FUNCTION_BLOCK "SysPos"   // FB2010, FBD
TITLE = manage a standard positioning system
{ S7_Optimized_Access := 'TRUE' }
AUTHOR : MiCROTEC
VERSION : 1.2
// -2017.03 : Martin
// stored: AutoNumber false, MemoryReserve 100, SetENOAutomatically false
   VAR_INPUT
      actual { ExternalAccessible := 'False'; ExternalVisible := 'False'; ExternalWritable := 'False'} : Real;   // actual position
      target { ExternalAccessible := 'False'; ExternalVisible := 'False'; ExternalWritable := 'False'} : Real;   // target position , start new position only if target position change
      tarMinPos { ExternalAccessible := 'False'; ExternalVisible := 'False'; ExternalWritable := 'False'} : Real;   // target position minimum
      tarMaxPos { ExternalAccessible := 'False'; ExternalVisible := 'False'; ExternalWritable := 'False'} : Real;   // target position maximum
      tolerance { ExternalAccessible := 'False'; ExternalVisible := 'False'; ExternalWritable := 'False'} : Real;   // tolerance for output signal position ok
      regPoint { ExternalAccessible := 'False'; ExternalVisible := 'False'; ExternalWritable := 'False'} : Real;   // regulation point (stop point before target position)
      regOn { ExternalAccessible := 'False'; ExternalVisible := 'False'; ExternalWritable := 'False'} : Bool;   // continuouse regulation on
      restart { ExternalAccessible := 'False'; ExternalVisible := 'False'; ExternalWritable := 'False'} : Bool;   // restart new positioning
      auto { ExternalAccessible := 'False'; ExternalVisible := 'False'; ExternalWritable := 'False'} : Bool;   // automatic (manP/manM and gain works only if auto is on)
      manP { ExternalAccessible := 'False'; ExternalVisible := 'False'; ExternalWritable := 'False'} : Bool;   // manual button plus
      manM { ExternalAccessible := 'False'; ExternalVisible := 'False'; ExternalWritable := 'False'} : Bool;   // manual button minus
      manPValue { ExternalAccessible := 'False'; ExternalVisible := 'False'; ExternalWritable := 'False'} : Real := 10.0;   // increase value in hand mode
      manMValue { ExternalAccessible := 'False'; ExternalVisible := 'False'; ExternalWritable := 'False'} : Real := 10.0;   // decrease value in hand mode
      stopRamp { ExternalAccessible := 'False'; ExternalVisible := 'False'; ExternalWritable := 'False'} : Real;   // position for stopramp
      stopSpeed { ExternalAccessible := 'False'; ExternalVisible := 'False'; ExternalWritable := 'False'} : Real;   // minimum speed for stopramp [0.0-1.0]
      approachPoint { ExternalAccessible := 'False'; ExternalVisible := 'False'; ExternalWritable := 'False'} : Real;   // aproach point, if its 0 than its OFF
   END_VAR
   VAR_OUTPUT
      plus { ExternalAccessible := 'False'; ExternalVisible := 'False'; ExternalWritable := 'False'} : Bool;   // command plus
      minus { ExternalAccessible := 'False'; ExternalVisible := 'False'; ExternalWritable := 'False'} : Bool;   // command minus
      slow { ExternalAccessible := 'False'; ExternalVisible := 'False'; ExternalWritable := 'False'} : Bool;   // slow
      posOk { ExternalAccessible := 'False'; ExternalVisible := 'False'; ExternalWritable := 'False'} : Bool;   // position ok
      tar { ExternalAccessible := 'False'; ExternalVisible := 'False'; ExternalWritable := 'False'} : Real;   // target position
      speedGain { ExternalAccessible := 'False'; ExternalVisible := 'False'; ExternalWritable := 'False'} : Real;   // gain for speed regulation ["StopSpeed" to 1.0]
   END_VAR
   VAR_IN_OUT
      Enc : "TypeEncoder";
   END_VAR
   VAR
      var { ExternalAccessible := 'False'; ExternalVisible := 'False'; ExternalWritable := 'False'} : Struct
         "bool" : Bool;
         "byte" : Byte;
         "word" : Word;
         "dword" : DWord;
         "int" : Int;
         "dint" : DInt;
         "real" : Real;
         s5time : S5Time;
         "time" : Time;
         hm : Array[1..16] of Bool;
         fm : Array[1..16] of Bool;
      END_STRUCT;
      statTargetOld { ExternalAccessible := 'False'; ExternalVisible := 'False'; ExternalWritable := 'False'} : Real;
      statApproachPoint { ExternalAccessible := 'False'; ExternalVisible := 'False'; ExternalWritable := 'False'} : Real;
      statRegPlusPos { ExternalAccessible := 'False'; ExternalVisible := 'False'; ExternalWritable := 'False'} : Real;
      statRegMinusPos { ExternalAccessible := 'False'; ExternalVisible := 'False'; ExternalWritable := 'False'} : Real;
      statInTolerance { ExternalAccessible := 'False'; ExternalVisible := 'False'; ExternalWritable := 'False'} : Bool;
      statAproachRun { ExternalAccessible := 'False'; ExternalVisible := 'False'; ExternalWritable := 'False'} : Bool;
      StatPosOk { ExternalAccessible := 'False'; ExternalVisible := 'False'; ExternalWritable := 'False'} : Bool;
      statSpeedDelta { ExternalAccessible := 'False'; ExternalVisible := 'False'; ExternalWritable := 'False'} : Real;
      statSpeedPerMm { ExternalAccessible := 'False'; ExternalVisible := 'False'; ExternalWritable := 'False'} : Real;
      statTarMin { ExternalAccessible := 'False'; ExternalVisible := 'False'; ExternalWritable := 'False'} : Bool;
      statTarMax { ExternalAccessible := 'False'; ExternalVisible := 'False'; ExternalWritable := 'False'} : Bool;
      statTar { ExternalAccessible := 'False'; ExternalVisible := 'False'; ExternalWritable := 'False'} : Real;
      statPlus { ExternalAccessible := 'False'; ExternalVisible := 'False'; ExternalWritable := 'False'} : Bool;
      statMinus { ExternalAccessible := 'False'; ExternalVisible := 'False'; ExternalWritable := 'False'} : Bool;
      statSpeedGain { ExternalAccessible := 'False'; ExternalVisible := 'False'; ExternalWritable := 'False'} : Real;
      statSlow { ExternalAccessible := 'False'; ExternalVisible := 'False'; ExternalWritable := 'False'} : Bool;
      statTarMaxPosOld : Real;
      statTarMinPosOld : Real;
   END_VAR
   VAR_TEMP   // added for the SCL form of the ladder/FBD networks
      _w1 : Bool;
      _w2 : Bool;
      _w3 : Bool;
   END_VAR
BEGIN

REGION Network 1: manual change target position
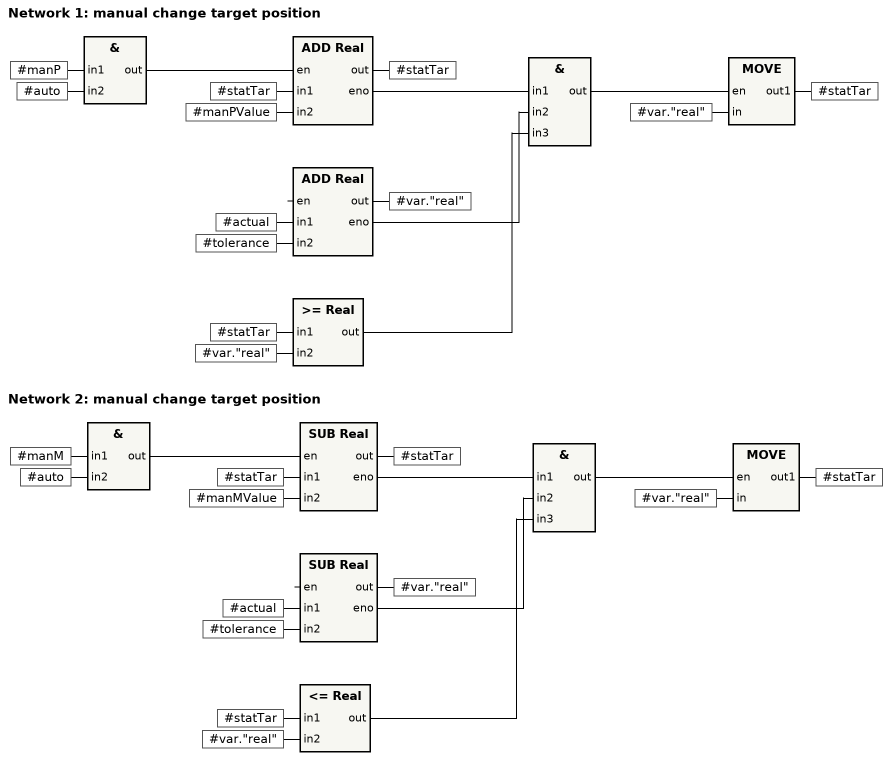
   // ENO of a box is taken as its EN; it also drops when the box reports an error
   #_w1 := #manP AND #auto;
   IF #_w1 THEN #statTar := #statTar + #manPValue; END_IF;
   #var."real" := #actual + #tolerance;
   IF #_w1 AND (#statTar >= #var."real") THEN #statTar := #var."real"; END_IF;
END_REGION

REGION Network 2: manual change target position
   // ENO of a box is taken as its EN; it also drops when the box reports an error
   #_w1 := #manM AND #auto;
   IF #_w1 THEN #statTar := #statTar - #manMValue; END_IF;
   #var."real" := #actual - #tolerance;
   IF #_w1 AND (#statTar <= #var."real") THEN #statTar := #var."real"; END_IF;
END_REGION

REGION Network 3: start positioning
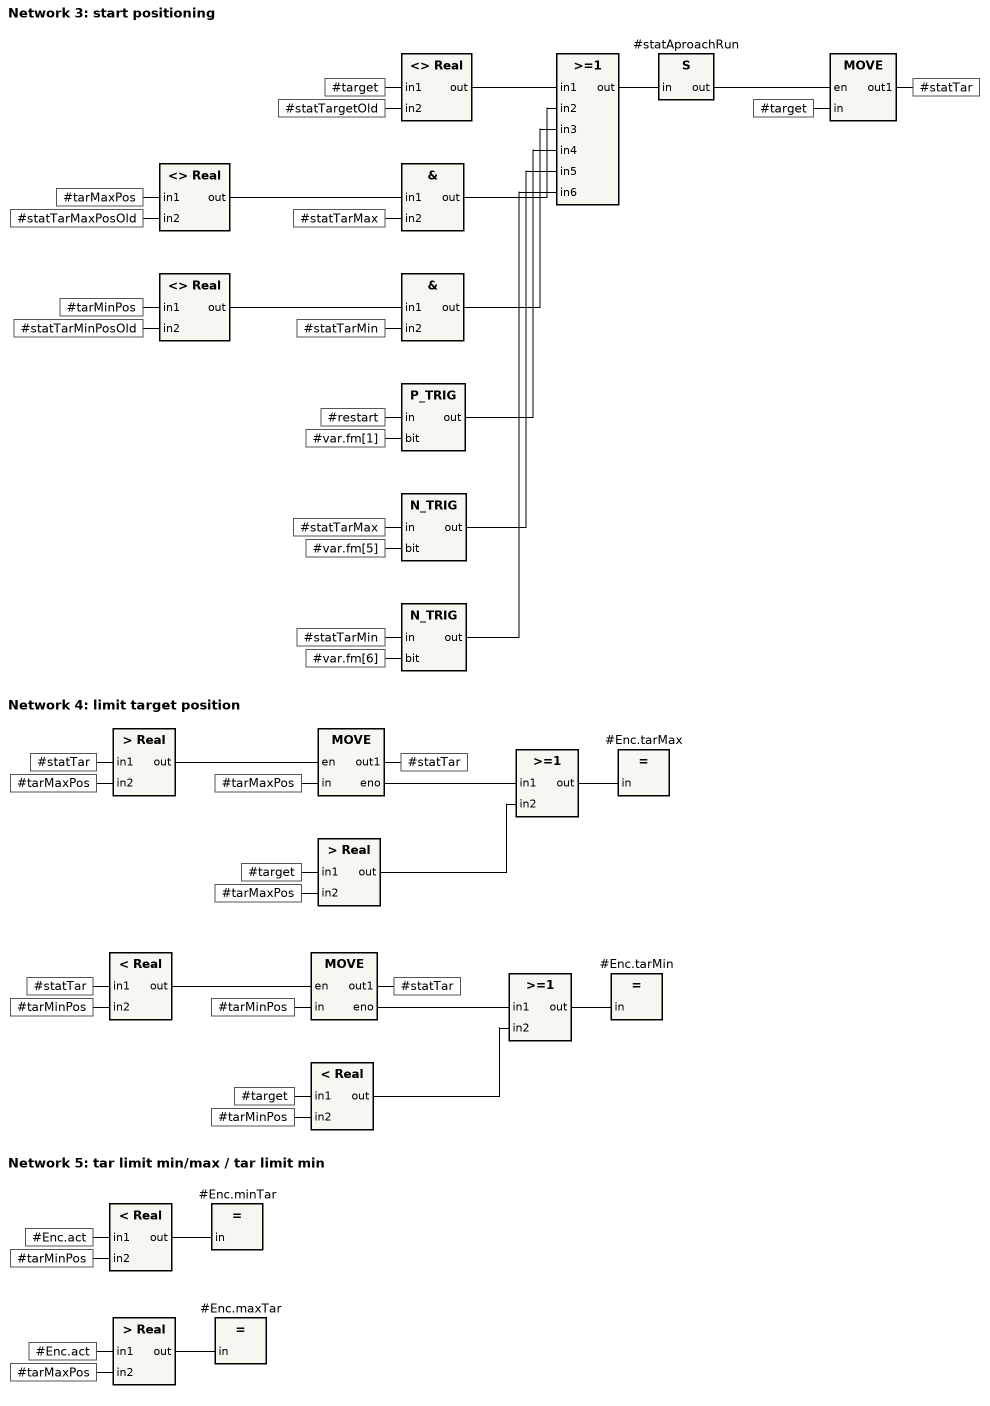
   #_w1 := #restart AND NOT #var.fm[1];   // rising edge
   #var.fm[1] := #restart;
   #_w2 := NOT #statTarMax AND #var.fm[5];   // falling edge
   #var.fm[5] := #statTarMax;
   #_w3 := NOT #statTarMin AND #var.fm[6];   // falling edge
   #var.fm[6] := #statTarMin;
   IF (#target <> #statTargetOld) OR ((#tarMaxPos <> #statTarMaxPosOld) AND #statTarMax) OR ((#tarMinPos <> #statTarMinPosOld) AND #statTarMin) OR #_w1 OR #_w2 OR #_w3 THEN
       #statAproachRun := TRUE;
       #statTar := #target;
   END_IF;
END_REGION

REGION Network 4: limit target position
   // ENO of a box is taken as its EN; it also drops when the box reports an error
   #_w1 := #statTar > #tarMaxPos;
   IF #_w1 THEN #statTar := #tarMaxPos; END_IF;
   #Enc.tarMax := #_w1 OR (#target > #tarMaxPos);
   #_w2 := #statTar < #tarMinPos;
   IF #_w2 THEN #statTar := #tarMinPos; END_IF;
   #Enc.tarMin := #_w2 OR (#target < #tarMinPos);
END_REGION

REGION Network 5: tar limit min/max / tar limit min
   #Enc.minTar := #Enc.act < #tarMinPos;
   #Enc.maxTar := #Enc.act > #tarMaxPos;
END_REGION

REGION Network 6 (SCL): approach/regulation point
   #statApproachPoint := #statTar + #approachPoint;

   #statRegMinusPos := #statTar - #regPoint;
   #statRegPlusPos := #statTar + #regPoint;
END_REGION

REGION Network 7: approachpoint reach
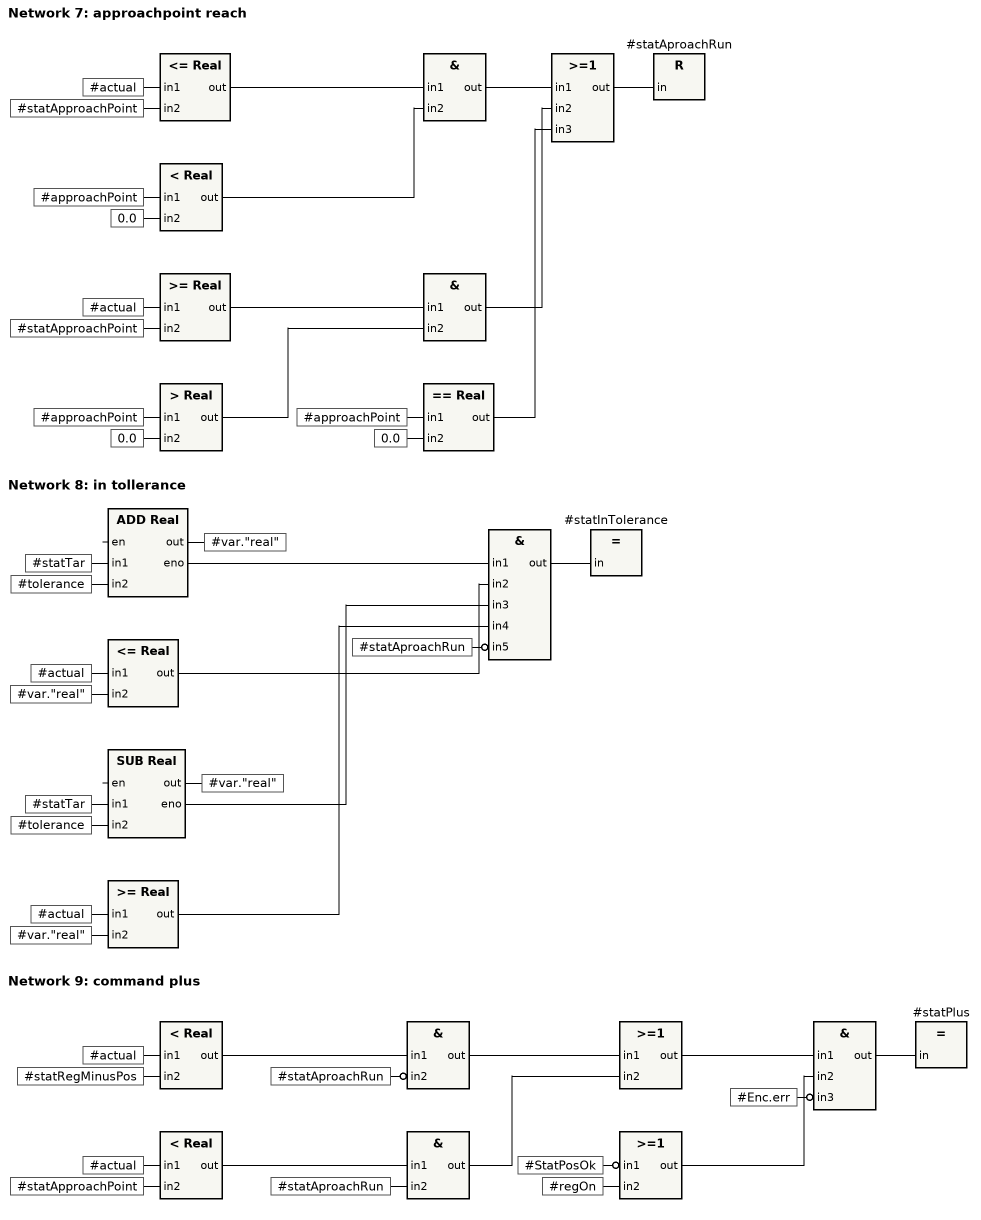
   IF ((#actual <= #statApproachPoint) AND (#approachPoint < 0.0)) OR ((#actual >= #statApproachPoint) AND (#approachPoint > 0.0)) OR (#approachPoint = 0.0) THEN
       #statAproachRun := FALSE;
   END_IF;
END_REGION

REGION Network 8: in tollerance
   // ENO of a box is taken as its EN; it also drops when the box reports an error
   #var."real" := #statTar + #tolerance;
   #_w1 := #actual <= #var."real";
   #var."real" := #statTar - #tolerance;
   #statInTolerance := #_w1 AND (#actual >= #var."real") AND NOT #statAproachRun;
END_REGION

REGION Network 9: command plus
   #statPlus := (((#actual < #statRegMinusPos) AND NOT #statAproachRun) OR ((#actual < #statApproachPoint) AND #statAproachRun)) AND (NOT #StatPosOk OR #regOn) AND NOT #Enc.err;
END_REGION

REGION Network 10: command minus
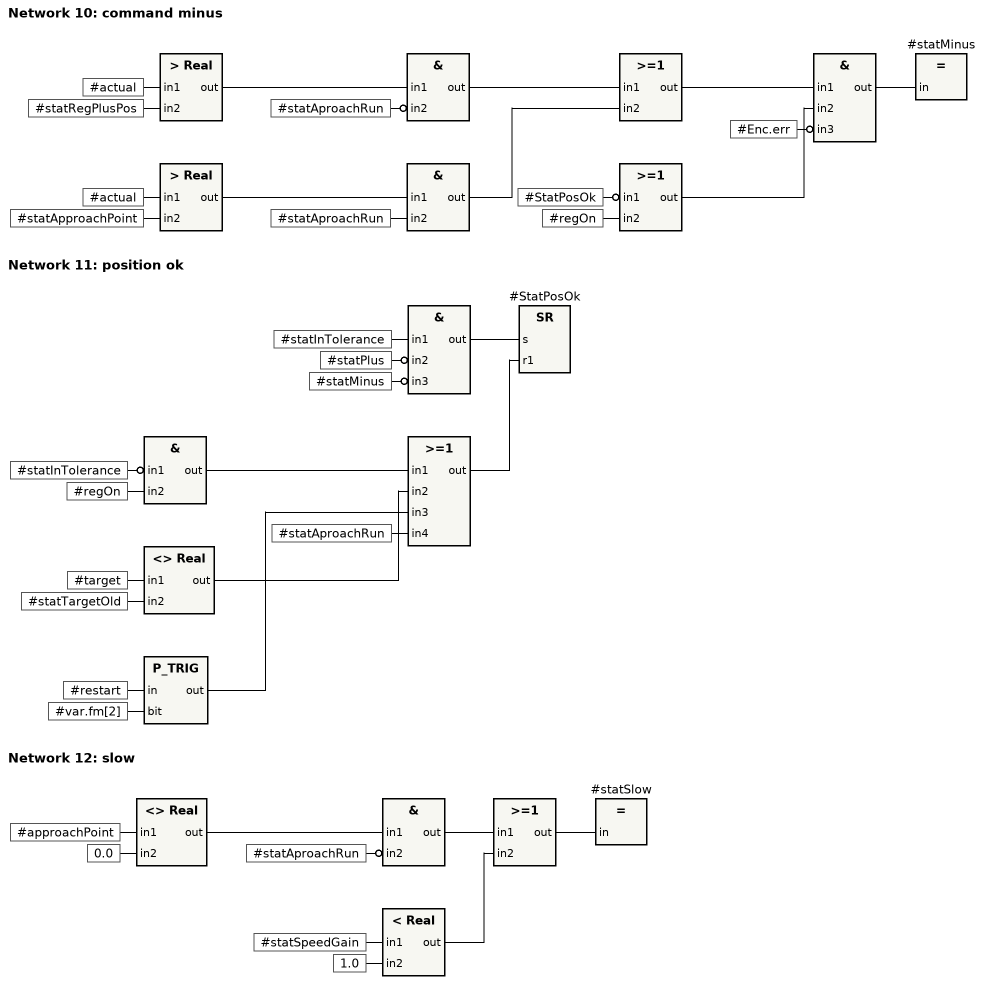
   #statMinus := (((#actual > #statRegPlusPos) AND NOT #statAproachRun) OR ((#actual > #statApproachPoint) AND #statAproachRun)) AND (NOT #StatPosOk OR #regOn) AND NOT #Enc.err;
END_REGION

REGION Network 11: position ok
   #_w1 := #restart AND NOT #var.fm[2];   // rising edge
   #var.fm[2] := #restart;
   IF #statInTolerance AND NOT #statPlus AND NOT #statMinus THEN
       #StatPosOk := TRUE;   // SR flip-flop
   END_IF;
   IF (NOT #statInTolerance AND #regOn) OR (#target <> #statTargetOld) OR #_w1 OR #statAproachRun THEN
       #StatPosOk := FALSE;
   END_IF;
END_REGION

REGION Network 12: slow
   #statSlow := ((#approachPoint <> 0.0) AND NOT #statAproachRun) OR (#statSpeedGain < 1.0);
END_REGION

REGION Network 13 (SCL): old position
   #statTargetOld := #target;
   #statTarMaxPosOld := #tarMaxPos;
   #statTarMinPosOld := #tarMinPos;
END_REGION

REGION Network 14 (SCL): speed gain for stop ramp
   #statSpeedDelta := 1.0 - #stopSpeed;
   #statSpeedPerMm := #statSpeedDelta / #stopRamp;
   #statSpeedGain := #stopSpeed + ABS_REAL((#statTar - #actual) * #statSpeedPerMm);

   IF #statSpeedGain < #stopSpeed THEN
       #statSpeedGain := #stopSpeed;
   END_IF;

   IF #statSpeedGain > 1.0 OR NOT #auto THEN
       #statSpeedGain := 1.0;
   END_IF;
END_REGION

REGION Network 15 (SCL): write outputs
       #plus := #statPlus;
       #minus := #statMinus;
       #slow:= #statSlow;
       #posOk := #StatPosOk;
       #tar := #statTar;
       #speedGain := #statSpeedGain;
END_REGION

REGION Network 16 (SCL): in/out data
       #Enc.tarMinPos := #tarMinPos;
       #Enc.tarMaxPos := #tarMaxPos;
       #Enc.act := #actual;
       #Enc.tar := #statTar;
       #Enc.posOk := #StatPosOk;
END_REGION
END_FUNCTION_BLOCK

FUNCTION_BLOCK "SysMotor"   // FB2060, FBD
TITLE = manage a motor with contactor equipment
{ S7_Optimized_Access := 'TRUE' }
AUTHOR : MiCROTEC
VERSION : 1.6
// -2017.03 : Martin
// stored: AutoNumber false, MemoryReserve 100, SetENOAutomatically false
   VAR_INPUT
      area { ExternalAccessible := 'False'; ExternalVisible := 'False'; ExternalWritable := 'False'} : Bool;   // 1=safety area on
      auto { ExternalAccessible := 'False'; ExternalVisible := 'False'; ExternalWritable := 'False'} : Bool;   // automatic
      manP { ExternalAccessible := 'False'; ExternalVisible := 'False'; ExternalWritable := 'False'} : Bool;   // manual plus
      manM { ExternalAccessible := 'False'; ExternalVisible := 'False'; ExternalWritable := 'False'} : Bool;   // manual minus
      autoP { ExternalAccessible := 'False'; ExternalVisible := 'False'; ExternalWritable := 'False'} : Bool;   // automatic plus
      autoM { ExternalAccessible := 'False'; ExternalVisible := 'False'; ExternalWritable := 'False'} : Bool;   // automatic minus
      ack { ExternalAccessible := 'False'; ExternalVisible := 'False'; ExternalWritable := 'False'} : Bool;   // fault acknowledge
      lampTest { ExternalAccessible := 'False'; ExternalVisible := 'False'; ExternalWritable := 'False'} : Bool;   // lamptest
      enableP { ExternalAccessible := 'False'; ExternalVisible := 'False'; ExternalWritable := 'False'} : Bool;   // release plus
      enableM { ExternalAccessible := 'False'; ExternalVisible := 'False'; ExternalWritable := 'False'} : Bool;   // release minus
      enAutoP { ExternalAccessible := 'False'; ExternalVisible := 'False'; ExternalWritable := 'False'} : Bool;   // release automatic plus
      enAutoM { ExternalAccessible := 'False'; ExternalVisible := 'False'; ExternalWritable := 'False'} : Bool;   // release automatic minus
      mpMotor { ExternalAccessible := 'False'; ExternalVisible := 'False'; ExternalWritable := 'False'} : Bool;   // 1=motor protection switch ok
      mpBrake { ExternalAccessible := 'False'; ExternalVisible := 'False'; ExternalWritable := 'False'} : Bool;   // 1=motor protection switch brake ok
      mpBrake2 { ExternalAccessible := 'False'; ExternalVisible := 'False'; ExternalWritable := 'False'} : Bool;   // 1=motor protection switch brake ok
      mpFan { ExternalAccessible := 'False'; ExternalVisible := 'False'; ExternalWritable := 'False'} : Bool;   // 1=motor protection switch fan ok
      thMotor { ExternalAccessible := 'False'; ExternalVisible := 'False'; ExternalWritable := 'False'} : Bool;   // 1=thermal contact motor ok
      thMotorRtd { ExternalAccessible := 'False'; ExternalVisible := 'False'; ExternalWritable := 'False'} : Int;   // thermal contact motor AE 8xRTD
      mSwitch { ExternalAccessible := 'False'; ExternalVisible := 'False'; ExternalWritable := 'False'} : Bool;   // 1=maintenance switch is ok
      fdb { ExternalAccessible := 'False'; ExternalVisible := 'False'; ExternalWritable := 'False'} : Bool;   // 1=feedback circuit ok
      changeDirTime { ExternalAccessible := 'False'; ExternalVisible := 'False'; ExternalWritable := 'False'} : Time := T#500MS;   // time wait to restart in oder direction
      restartTime { ExternalAccessible := 'False'; ExternalVisible := 'False'; ExternalWritable := 'False'} : Time := T#500MS;   // time wait to restart in any direction
      brakeOnTime { ExternalAccessible := 'False'; ExternalVisible := 'False'; ExternalWritable := 'False'} : Time := T#10MS;   // time wait to open the brake
      brakeOffTime { ExternalAccessible := 'False'; ExternalVisible := 'False'; ExternalWritable := 'False'} : Time := T#10MS;   // time wait to close the brake
      metPerMin { ExternalAccessible := 'False'; ExternalVisible := 'False'; ExternalWritable := 'False'} : Real := 1.0;   // meter per minute with nominal speed
      cycle { ExternalAccessible := 'False'; ExternalVisible := 'False'; ExternalWritable := 'False'} : Real;   // cycle
   END_VAR
   VAR_OUTPUT
      plus { ExternalAccessible := 'False'; ExternalVisible := 'False'; ExternalWritable := 'False'} : Bool;   // drive plus
      minus { ExternalAccessible := 'False'; ExternalVisible := 'False'; ExternalWritable := 'False'} : Bool;   // drive minus
      brake { ExternalAccessible := 'False'; ExternalVisible := 'False'; ExternalWritable := 'False'} : Bool;   // brake open
      brake2 { ExternalAccessible := 'False'; ExternalVisible := 'False'; ExternalWritable := 'False'} : Bool;   // brake open
      enStartP { ExternalAccessible := 'False'; ExternalVisible := 'False'; ExternalWritable := 'False'} : Bool;   // release drive plus
      enStartM { ExternalAccessible := 'False'; ExternalVisible := 'False'; ExternalWritable := 'False'} : Bool;   // release drive minus
      fan { ExternalAccessible := 'False'; ExternalVisible := 'False'; ExternalWritable := 'False'} : Bool;   // fan on
      lamp { ExternalAccessible := 'False'; ExternalVisible := 'False'; ExternalWritable := 'False'} : Bool;   // indication lamp
      lamp2 { ExternalAccessible := 'False'; ExternalVisible := 'False'; ExternalWritable := 'False'} : Bool;   // indication lamp 2
      actSpeed { ExternalAccessible := 'False'; ExternalVisible := 'False'; ExternalWritable := 'False'} : Real;   // actual speed
      mmCycle { ExternalAccessible := 'False'; ExternalVisible := 'False'; ExternalWritable := 'False'} : Real;   // milimeter per cycle
      err { ExternalAccessible := 'False'; ExternalVisible := 'False'; ExternalWritable := 'False'} : Bool;   // fault
   END_VAR
   VAR_IN_OUT
      Mot : "TypeMotor";   // Daten an VISU Motor
   END_VAR
   VAR
      var { ExternalAccessible := 'False'; ExternalVisible := 'False'; ExternalWritable := 'False'} : Struct
         true : Bool;
         false : Bool;
         "bool" : Bool;
         "byte" : Byte;
         "word" : Word;
         "dword" : DWord;
         "int" : Int;
         "dint" : DInt;
         "real" : Real;
         s5time : S5Time;
         "time" : Time;
         hm : Array[1..50] of Bool;
         fm : Array[1..50] of Bool;
      END_STRUCT;
      T { ExternalAccessible := 'False'; ExternalVisible := 'False'; ExternalWritable := 'False'} : Array[1..15] of IEC_TIMER;
      restartBreak { ExternalAccessible := 'False'; ExternalVisible := 'False'; ExternalWritable := 'False'} : Bool;
      man { ExternalAccessible := 'False'; ExternalVisible := 'False'; ExternalWritable := 'False'} : Bool;
      changeDirDelM { ExternalAccessible := 'False'; ExternalVisible := 'False'; ExternalWritable := 'False'} : Bool;
      changeDirDelP { ExternalAccessible := 'False'; ExternalVisible := 'False'; ExternalWritable := 'False'} : Bool;
      mpFanOffDel { ExternalAccessible := 'False'; ExternalVisible := 'False'; ExternalWritable := 'False'} : Bool;
      brakeOnDel { ExternalAccessible := 'False'; ExternalVisible := 'False'; ExternalWritable := 'False'} : Bool;
      brakeOffDel { ExternalAccessible := 'False'; ExternalVisible := 'False'; ExternalWritable := 'False'} : Bool;
      autoOld { ExternalAccessible := 'False'; ExternalVisible := 'False'; ExternalWritable := 'False'} : Bool;
   END_VAR
   VAR_TEMP
      tempAck : Bool;
   END_VAR
   VAR_TEMP   // added for the SCL form of the ladder/FBD networks
      _w1 : Bool;
      _w2 : Bool;
   END_VAR
BEGIN

REGION Network 1: ack
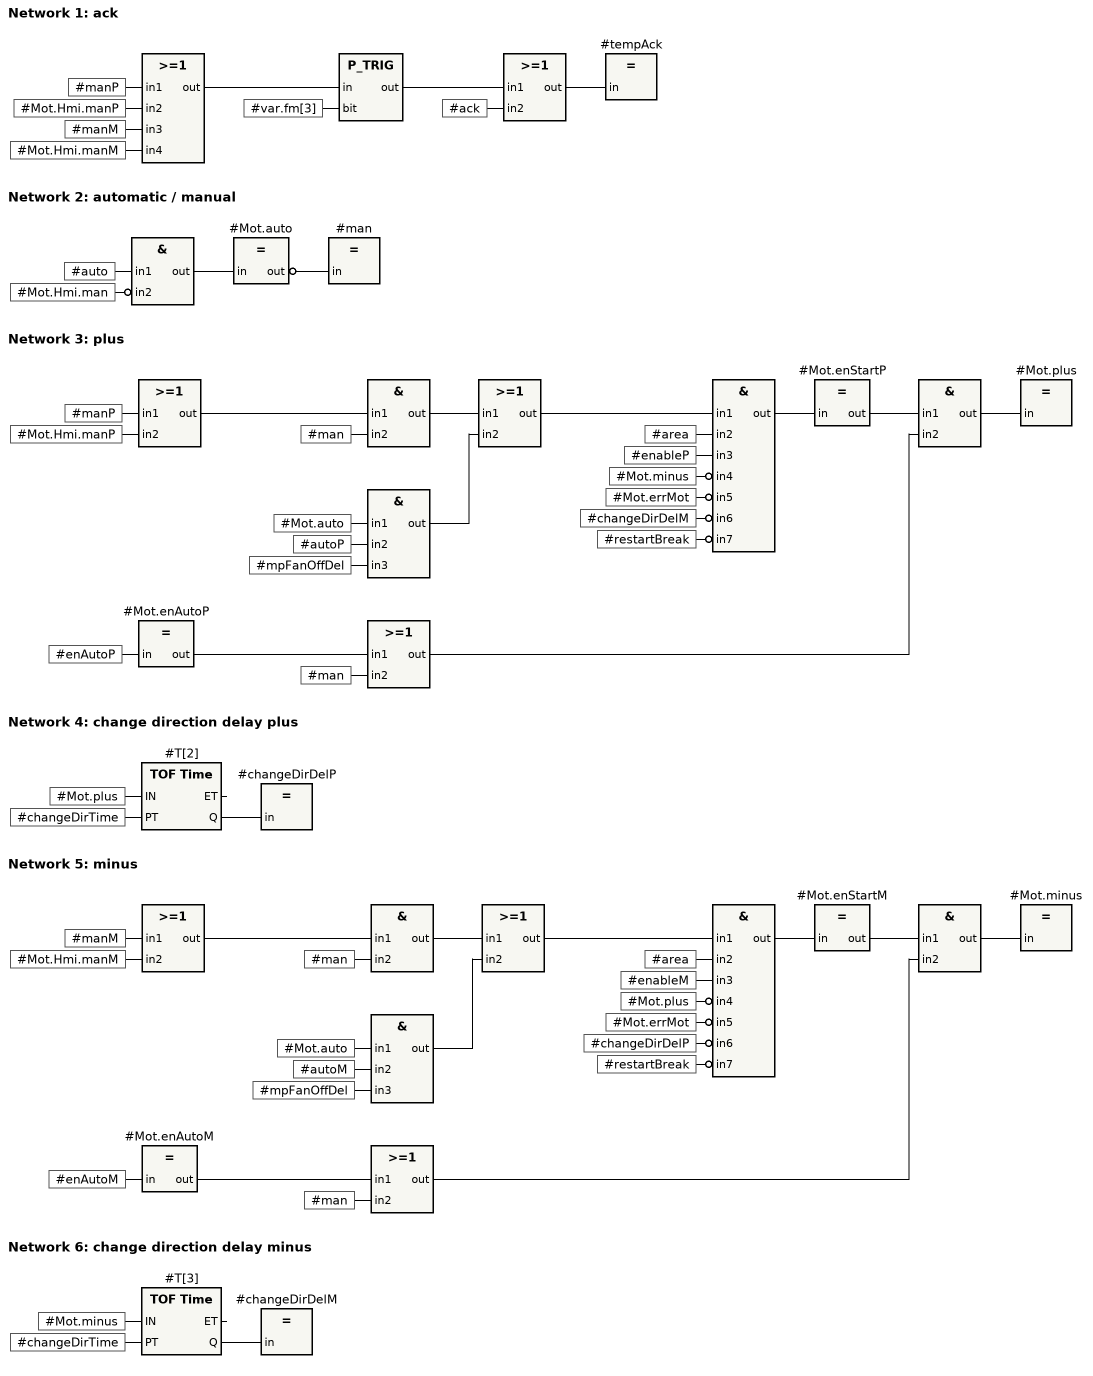
   #_w1 := #manP OR #Mot.Hmi.manP OR #manM OR #Mot.Hmi.manM;
   #_w2 := #_w1 AND NOT #var.fm[3];   // rising edge
   #var.fm[3] := #_w1;
   #tempAck := #_w2 OR #ack;
END_REGION

REGION Network 2: automatic / manual
   #_w1 := #auto AND NOT #Mot.Hmi.man;
   #Mot.auto := #_w1;
   #man := NOT #_w1;
END_REGION

REGION Network 3: plus
   #Mot.enStartP := (((#manP OR #Mot.Hmi.manP) AND #man) OR (#Mot.auto AND #autoP AND #mpFanOffDel)) AND #area AND #enableP AND NOT #Mot.minus AND NOT #Mot.errMot AND NOT #changeDirDelM AND NOT #restartBreak;
   #Mot.enAutoP := #enAutoP;
   #Mot.plus := #Mot.enStartP AND (#enAutoP OR #man);
END_REGION

REGION Network 4: change direction delay plus
   #T[2].TOF(IN := #Mot.plus, PT := #changeDirTime);
   #changeDirDelP := #T[2].Q;
END_REGION

REGION Network 5: minus
   #Mot.enStartM := (((#manM OR #Mot.Hmi.manM) AND #man) OR (#Mot.auto AND #autoM AND #mpFanOffDel)) AND #area AND #enableM AND NOT #Mot.plus AND NOT #Mot.errMot AND NOT #changeDirDelP AND NOT #restartBreak;
   #Mot.enAutoM := #enAutoM;
   #Mot.minus := #Mot.enStartM AND (#enAutoM OR #man);
END_REGION

REGION Network 6: change direction delay minus
   #T[3].TOF(IN := #Mot.minus, PT := #changeDirTime);
   #changeDirDelM := #T[3].Q;
END_REGION

REGION Network 7: restart delay
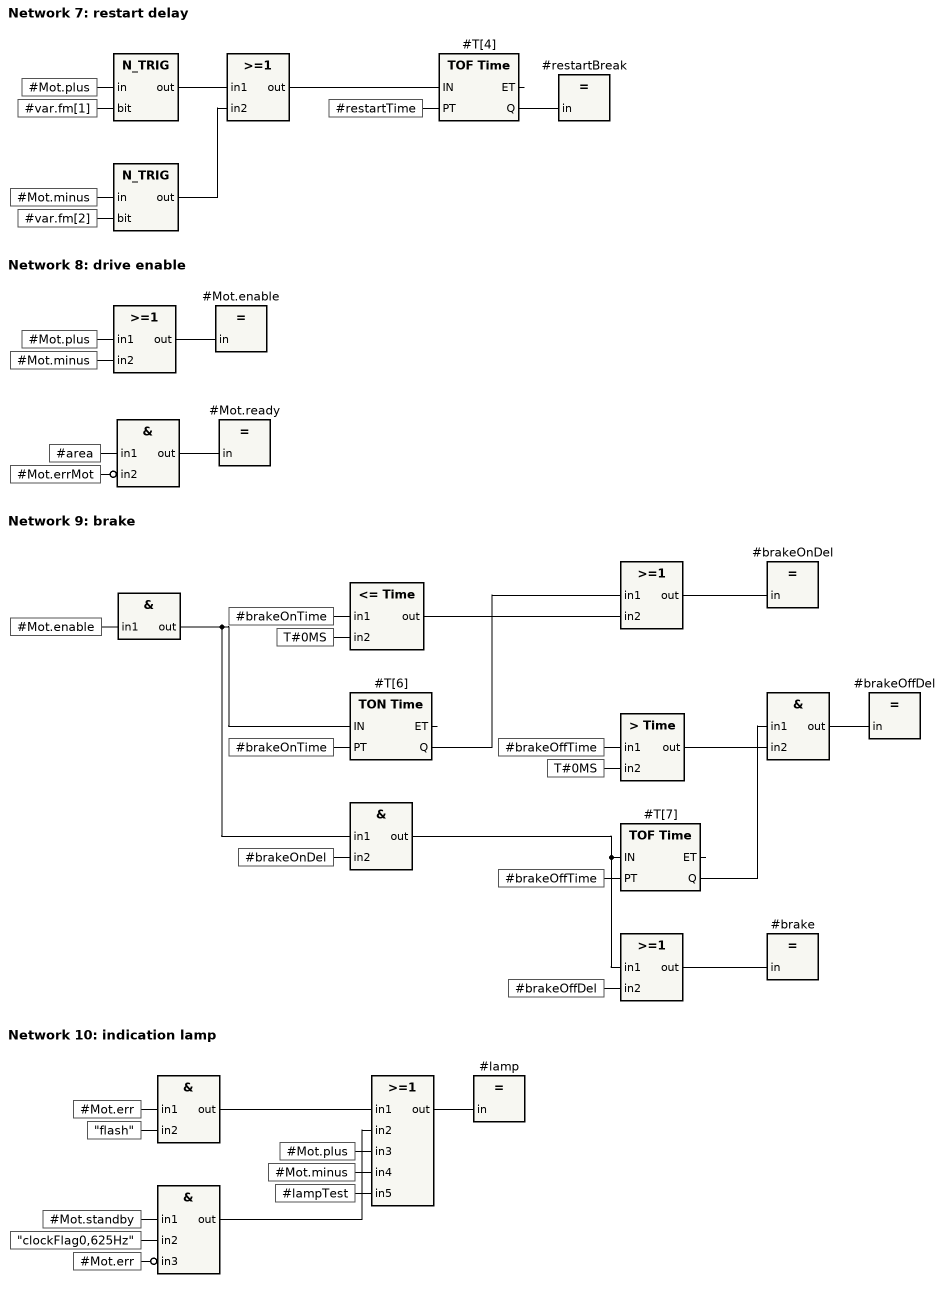
   #_w1 := NOT #Mot.plus AND #var.fm[1];   // falling edge
   #var.fm[1] := #Mot.plus;
   #_w2 := NOT #Mot.minus AND #var.fm[2];   // falling edge
   #var.fm[2] := #Mot.minus;
   #T[4].TOF(IN := #_w1 OR #_w2, PT := #restartTime);
   #restartBreak := #T[4].Q;
END_REGION

REGION Network 8: drive enable
   #Mot.enable := #Mot.plus OR #Mot.minus;
   #Mot.ready := #area AND NOT #Mot.errMot;
END_REGION

REGION Network 9: brake
   #T[6].TON(IN := #Mot.enable, PT := #brakeOnTime);
   #brakeOnDel := #T[6].Q OR (#brakeOnTime <= T#0MS);
   #_w1 := #Mot.enable AND #brakeOnDel;
   #T[7].TOF(IN := #_w1, PT := #brakeOffTime);
   #brakeOffDel := #T[7].Q AND (#brakeOffTime > T#0MS);
   #brake := #_w1 OR #brakeOffDel;
END_REGION

REGION Network 10: indication lamp
   #lamp := (#Mot.err AND "flash") OR (#Mot.standby AND "clockFlag0,625Hz" AND NOT #Mot.err) OR #Mot.plus OR #Mot.minus OR #lampTest;
END_REGION

REGION Network 11: direction plus delayed
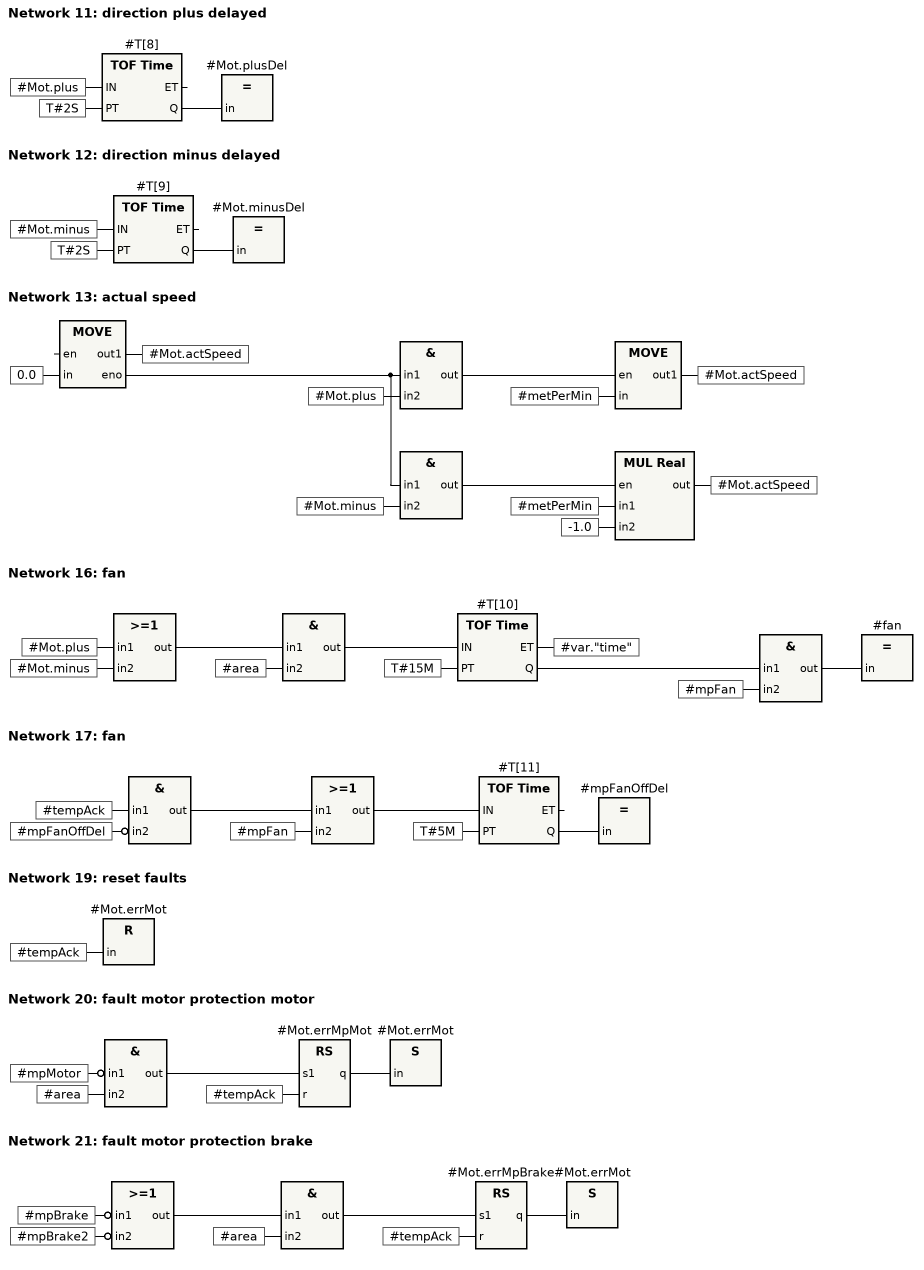
   #T[8].TOF(IN := #Mot.plus, PT := T#2S);
   #Mot.plusDel := #T[8].Q;
END_REGION

REGION Network 12: direction minus delayed
   #T[9].TOF(IN := #Mot.minus, PT := T#2S);
   #Mot.minusDel := #T[9].Q;
END_REGION

REGION Network 13: actual speed
   // ENO of a box is taken as its EN; it also drops when the box reports an error
   #Mot.actSpeed := 0.0;
   IF #Mot.plus THEN #Mot.actSpeed := #metPerMin; END_IF;
   IF #Mot.minus THEN #Mot.actSpeed := #metPerMin * (-1.0); END_IF;
END_REGION

REGION Network 14 (SCL): millimeter per cycle
   #Mot.mmCycle := 0.0;
   IF #Mot.plus OR #Mot.minus THEN
      #Mot.mmCycle := (#cycle *  #Mot.actSpeed ) / 60.0;
   END_IF;
END_REGION

REGION Network 15: -- fan--
END_REGION

REGION Network 16: fan
   #T[10].TOF(IN := (#Mot.plus OR #Mot.minus) AND #area, PT := T#15M, ET => #var."time");
   #fan := #T[10].Q AND #mpFan;
END_REGION

REGION Network 17: fan
   #T[11].TOF(IN := (#tempAck AND NOT #mpFanOffDel) OR #mpFan, PT := T#5M);
   #mpFanOffDel := #T[11].Q;
END_REGION

REGION Network 18: --faults--
END_REGION

REGION Network 19: reset faults
   IF #tempAck THEN #Mot.errMot := FALSE; END_IF;
END_REGION

REGION Network 20: fault motor protection motor
   IF #tempAck THEN
       #Mot.errMpMot := FALSE;   // RS flip-flop
   END_IF;
   IF NOT #mpMotor AND #area THEN #Mot.errMpMot := TRUE; END_IF;
   IF #Mot.errMpMot THEN #Mot.errMot := TRUE; END_IF;
END_REGION

REGION Network 21: fault motor protection brake
   IF #tempAck THEN
       #Mot.errMpBrake := FALSE;   // RS flip-flop
   END_IF;
   IF (NOT #mpBrake OR NOT #mpBrake2) AND #area THEN #Mot.errMpBrake := TRUE; END_IF;
   IF #Mot.errMpBrake THEN #Mot.errMot := TRUE; END_IF;
END_REGION

REGION Network 22: fault thermal contact motor
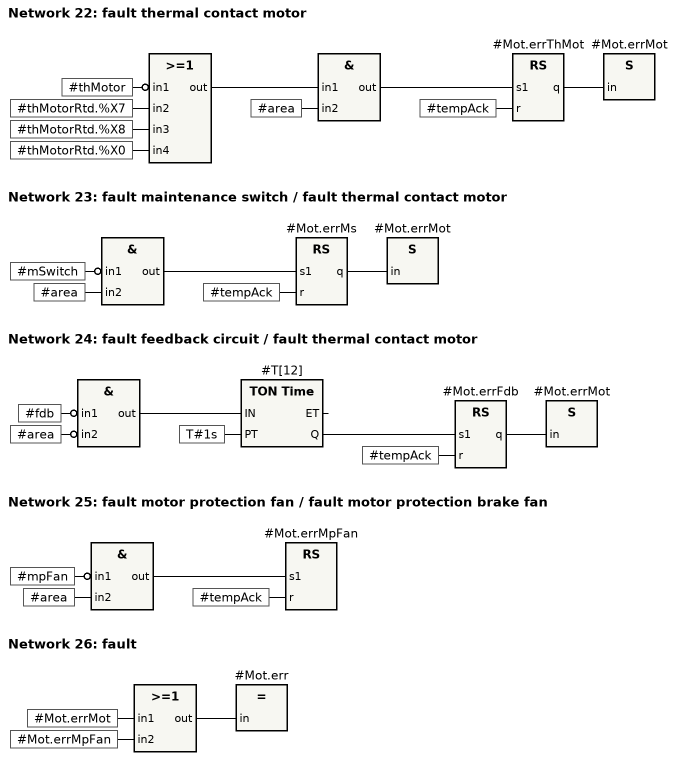
   IF #tempAck THEN
       #Mot.errThMot := FALSE;   // RS flip-flop
   END_IF;
   IF (NOT #thMotor OR #thMotorRtd.%X7 OR #thMotorRtd.%X8 OR #thMotorRtd.%X0) AND #area THEN
       #Mot.errThMot := TRUE;
   END_IF;
   IF #Mot.errThMot THEN #Mot.errMot := TRUE; END_IF;
END_REGION

REGION Network 23: fault maintenance switch / fault thermal contact motor
   IF #tempAck THEN
       #Mot.errMs := FALSE;   // RS flip-flop
   END_IF;
   IF NOT #mSwitch AND #area THEN #Mot.errMs := TRUE; END_IF;
   IF #Mot.errMs THEN #Mot.errMot := TRUE; END_IF;
END_REGION

REGION Network 24: fault feedback circuit / fault thermal contact motor
   #T[12].TON(IN := NOT #fdb AND NOT #area, PT := T#1s);
   IF #tempAck THEN
       #Mot.errFdb := FALSE;   // RS flip-flop
   END_IF;
   IF #T[12].Q THEN #Mot.errFdb := TRUE; END_IF;
   IF #Mot.errFdb THEN #Mot.errMot := TRUE; END_IF;
END_REGION

REGION Network 25: fault motor protection fan / fault motor protection brake fan
   IF #tempAck THEN
       #Mot.errMpFan := FALSE;   // RS flip-flop
   END_IF;
   IF NOT #mpFan AND #area THEN #Mot.errMpFan := TRUE; END_IF;
END_REGION

REGION Network 26: fault
   #Mot.err := #Mot.errMot OR #Mot.errMpFan;
END_REGION

REGION Network 27 (SCL): write outputs
      #plus := #Mot.plus;
      #minus := #Mot.minus;
      #brake2 := #brake;
      #enStartP :=  #Mot.enStartP ;
      #enStartM :=  #Mot.enStartM;
      #lamp2 :=#lamp;
      #err :=  #Mot.err;
      #actSpeed :=  #Mot.actSpeed ;
      #mmCycle := #Mot.mmCycle;
END_REGION

REGION Network 28 (SCL): in/out data
      #Mot.run := #Mot.plus OR #Mot.minus;
      #Mot.runDel :=  #Mot.plusDel  OR  #Mot.minusDel ;
      #Mot.errNr := 0;
      #Mot.tarSpeed := #metPerMin;
      #Mot.area := #area;

       IF #auto AND NOT #autoOld THEN
           #Mot.Hmi.man := false;
           #Mot.Hmi.manP := false;
           #Mot.Hmi.manM := false;
       END_IF;
       #autoOld := #auto;
END_REGION
END_FUNCTION_BLOCK

FUNCTION_BLOCK "AdjTop"   // FB520, FBD
{ S7_Optimized_Access := 'TRUE' }
// stored: AutoNumber false, MemoryReserve 100, SetENOAutomatically false
   VAR
      Var { ExternalAccessible := 'False'; ExternalVisible := 'False'; ExternalWritable := 'False'} : "TypeVar";
      Cmd { ExternalAccessible := 'False'; ExternalVisible := 'False'; ExternalWritable := 'False'} : "TypeCmd";
      Enc { ExternalAccessible := 'False'; ExternalVisible := 'False'; ExternalWritable := 'False'} : "SysCounterFast";
      Pos { ExternalAccessible := 'False'; ExternalVisible := 'False'; ExternalWritable := 'False'} : "SysPos";
      AdjSlow { ExternalAccessible := 'False'; ExternalVisible := 'False'; ExternalWritable := 'False'} : "SysMotor";
      AdjFast { ExternalAccessible := 'False'; ExternalVisible := 'False'; ExternalWritable := 'False'} : "SysLinMotC1150";
      TAutoOn { ExternalAccessible := 'False'; ExternalVisible := 'False'; ExternalWritable := 'False'} : TON_TIME;
      TAutoTarPosManOn { ExternalAccessible := 'False'; ExternalVisible := 'False'; ExternalWritable := 'False'} : TON_TIME;
      T { ExternalAccessible := 'False'; ExternalVisible := 'False'; ExternalWritable := 'False'} : Array[1..5] of IEC_TIMER;
      adjFastPnSlaveOff { ExternalAccessible := 'False'; ExternalVisible := 'False'; ExternalWritable := 'False'} : "SysPnSlaveDeactivate";
      tarOld { ExternalAccessible := 'False'; ExternalVisible := 'False'; ExternalWritable := 'False'} : DInt;
      autoTarPosMan { ExternalAccessible := 'False'; ExternalVisible := 'False'; ExternalWritable := 'False'} : Bool;
      setValueEnc { ExternalAccessible := 'False'; ExternalVisible := 'False'; ExternalWritable := 'False'} : Bool;
      autoRef { ExternalAccessible := 'False'; ExternalVisible := 'False'; ExternalWritable := 'False'} : Bool;
   END_VAR
   VAR_TEMP
      CtrlPc : Struct
         ackErr : Bool;
         manModeActive : Bool;
         manP : Bool;
         manM : Bool;
         manRefRun : Bool;
      END_STRUCT;
      CtrlLinMot : Struct
         Mode : Int;
         Target : Real;
         Speed : Real;
         Acc : Real;
         Dec : Real;
         Jerk : Real;
      END_STRUCT;
      refPosDiff : DInt;
      offsetNoStd : Real;
      refPosDiffCalib : DInt;
      modeCalib : Int;
      disMechanicToZero : Int;   // distance mechanic part top to zero [mm]
   END_VAR
   VAR_TEMP   // added for the SCL form of the ladder/FBD networks
      _w1 : Bool;
   END_VAR
BEGIN

REGION Network 1 (SCL): offset for no standard calibration
   (* 
   normally the distance from camera to board should be 550mm
   for special application the distance is different
   the distance can be changed in the goldeneye program
   if its different then 550mm a offset will be added
   *) 

   #offsetNoStd := 0.0;
   IF "ComRd".Data.Top.RefPosToBoard <> 550 THEN
       #offsetNoStd := (DINT_TO_REAL("ComRd".Data.Top.RefPosToBoard) - 550.0);
   END_IF;
END_REGION

REGION Network 2 (SCL): calibration value for offset
   (* 
   modus for calibartion
   camera must be referenced first
   mode 1 -->   the camera must be moved manually to position 550mm from board and
                 then press "Set Nullpoint"
   mode 2 -->   the camera must be moved to a other position and
                 then must be measured from the calibration tool to the camera and
                 this value must be putted in after pressing "Set Nullpoint"
   *)        
   #disMechanicToZero := 963;

   #modeCalib := 2;
   IF #modeCalib = 1 THEN
       #refPosDiffCalib := "ComRd".Data.Top.TargetPos;
   ELSIF #modeCalib = 2 THEN
       #refPosDiffCalib := (#disMechanicToZero * 10) - ("ComRd".Data.Top.CalibratePos + 5500);
   END_IF;
END_REGION

REGION Network 3 (SCL): calibration value from pc
   "ComSd".Data.Top.SetCalibratePosOk := FALSE;

   IF "ComRd".Data.Top.SetCalibratePos THEN

       IF "G".Cfg.adjTopActive THEN
           "Ref".adjTopCalOffset  := REAL_TO_DINT("Enc"."8BC1.T".act * 10.0) - #refPosDiffCalib;
       ELSIF "G".Cfg.adjTopActiveLinMot THEN
           "Ref".adjTopCalOffset  := REAL_TO_DINT("Enc"."8U1.T".act * 10.0) - #refPosDiffCalib;
       END_IF;

       "ComSd".Data.Top.SetCalibratePosOk := TRUE;
   END_IF;
END_REGION

REGION Network 4 (SCL): target position
   #Cmd.target := "G".Batch.thickness;
   IF ("G".Cfg.modeDimension = 3 OR "G".Cfg.modeDimension = 4) AND NOT "G".Batch.stdActive THEN
       #Cmd.target := "G".Batch.thicknessMeasure;
   END_IF;

   IF #autoTarPosMan THEN
       #Cmd.target := DINT_TO_REAL(("ComRd".Data.Top.TargetPos)) / 10.0;
   END_IF;

   "Ref".adjTopTar := #Cmd.target + (DINT_TO_REAL("Ref".adjTopCalOffset) / 10.0) + #offsetNoStd;
END_REGION

REGION Network 5 (SCL): data from pc
   IF NOT "G".errComPc THEN
       #CtrlPc.manModeActive := "ComRd".Data.Top.ManModeActive;
       #CtrlPc.manP := "ComRd".Data.Top.ManPlus;
       #CtrlPc.manM := "ComRd".Data.Top.ManMinus;
       #CtrlPc.manRefRun := "ComRd".Data.Top.ManRefRun;
   ELSE
       #CtrlPc.manModeActive := TRUE;
       #CtrlPc.manP := FALSE;
       #CtrlPc.manM := FALSE;
       #CtrlPc.manRefRun := FALSE;
   END_IF;

   #CtrlPc.ackErr := "G".ack;
END_REGION

REGION Network 6: off
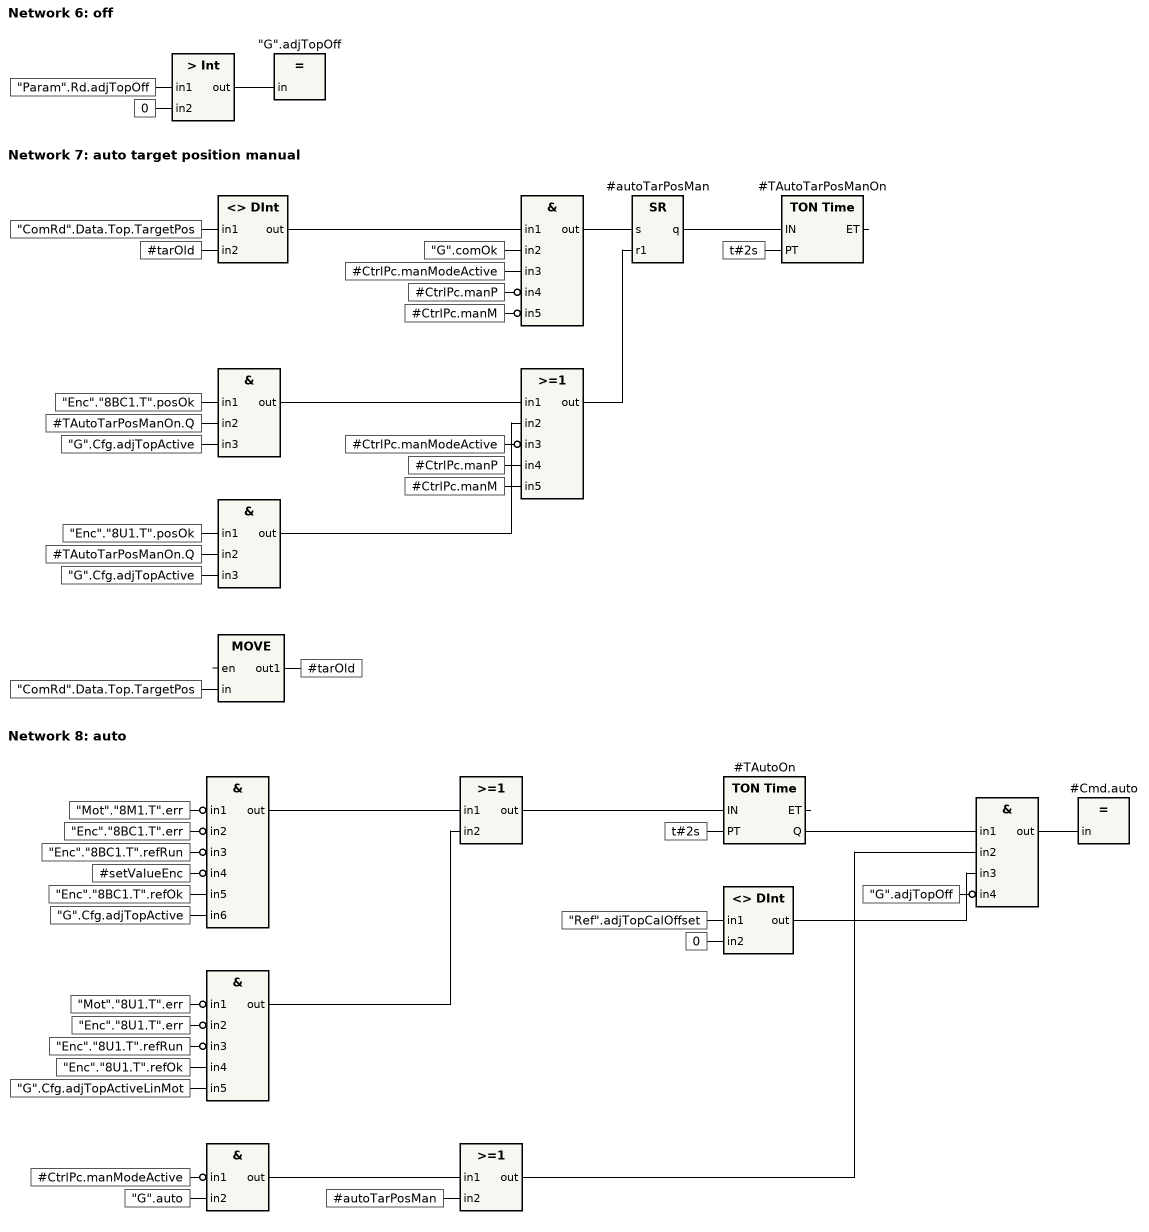
   "G".adjTopOff := "Param".Rd.adjTopOff > 0;
END_REGION

REGION Network 7: auto target position manual
   IF ("ComRd".Data.Top.TargetPos <> #tarOld) AND "G".comOk AND #CtrlPc.manModeActive AND NOT #CtrlPc.manP AND NOT #CtrlPc.manM THEN
       #autoTarPosMan := TRUE;   // SR flip-flop
   END_IF;
   IF ("Enc"."8BC1.T".posOk AND #TAutoTarPosManOn.Q AND "G".Cfg.adjTopActive) OR ("Enc"."8U1.T".posOk AND #TAutoTarPosManOn.Q AND "G".Cfg.adjTopActive) OR NOT #CtrlPc.manModeActive OR #CtrlPc.manP OR #CtrlPc.manM THEN
       #autoTarPosMan := FALSE;
   END_IF;
   #TAutoTarPosManOn(IN := #autoTarPosMan, PT := t#2s);   // TON
   #tarOld := "ComRd".Data.Top.TargetPos;
END_REGION

REGION Network 8: auto
   #TAutoOn(IN := (NOT "Mot"."8M1.T".err AND NOT "Enc"."8BC1.T".err AND NOT "Enc"."8BC1.T".refRun AND NOT #setValueEnc AND "Enc"."8BC1.T".refOk AND "G".Cfg.adjTopActive) OR (NOT "Mot"."8U1.T".err AND NOT "Enc"."8U1.T".err AND NOT "Enc"."8U1.T".refRun AND "Enc"."8U1.T".refOk AND "G".Cfg.adjTopActiveLinMot),   // TON
            PT := t#2s);
   #Cmd.auto := #TAutoOn.Q AND ((NOT #CtrlPc.manModeActive AND "G".auto) OR #autoTarPosMan) AND ("Ref".adjTopCalOffset <> 0) AND NOT "G".adjTopOff;
END_REGION

REGION Network 9: manual
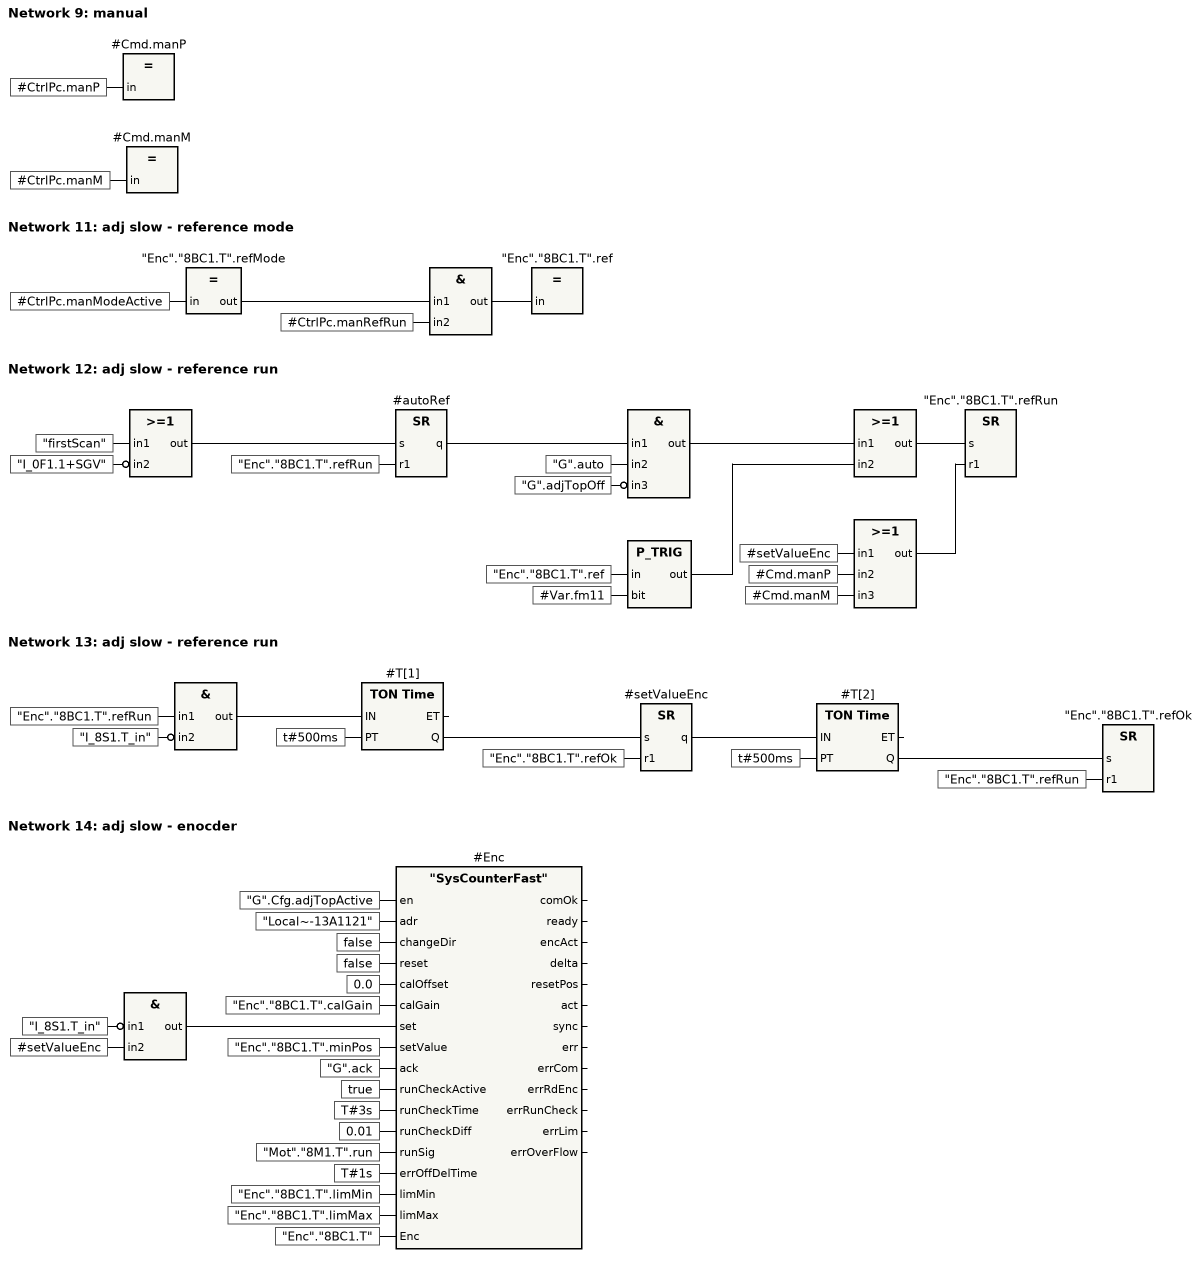
   #Cmd.manP := #CtrlPc.manP;
   #Cmd.manM := #CtrlPc.manM;
END_REGION

REGION Network 10 (SCL): adj slow - calibration value
   "Enc"."8BC1.T".calGain := -0.0275;

   "Enc"."8BC1.T".minPos := 10.0;
   "Enc"."8BC1.T".maxPos := 210.0;

   "Enc"."8BC1.T".limMin := "Enc"."8BC1.T".minPos - 5.0;
   "Enc"."8BC1.T".limMax := "Enc"."8BC1.T".maxPos + 5.0;

   "Enc"."8BC1.T".tarMinPos := "Enc"."8BC1.T".minPos + 0.0;
   "Enc"."8BC1.T".tarMaxPos := "Enc"."8BC1.T".maxPos - 0.0;
END_REGION

REGION Network 11: adj slow - reference mode
   "Enc"."8BC1.T".refMode := #CtrlPc.manModeActive;
   "Enc"."8BC1.T".ref := #CtrlPc.manModeActive AND #CtrlPc.manRefRun;
END_REGION

REGION Network 12: adj slow - reference run
   IF "firstScan" OR NOT "I_0F1.1+SGV" THEN
       #autoRef := TRUE;   // SR flip-flop
   END_IF;
   IF "Enc"."8BC1.T".refRun THEN #autoRef := FALSE; END_IF;
   #_w1 := "Enc"."8BC1.T".ref AND NOT #Var.fm11;   // rising edge
   #Var.fm11 := "Enc"."8BC1.T".ref;
   IF (#autoRef AND "G".auto AND NOT "G".adjTopOff) OR #_w1 THEN
       "Enc"."8BC1.T".refRun := TRUE;   // SR flip-flop
   END_IF;
   IF #setValueEnc OR #Cmd.manP OR #Cmd.manM THEN "Enc"."8BC1.T".refRun := FALSE; END_IF;
END_REGION

REGION Network 13: adj slow - reference run
   #T[1].TON(IN := "Enc"."8BC1.T".refRun AND NOT "I_8S1.T_in", PT := t#500ms);
   IF #T[1].Q THEN
       #setValueEnc := TRUE;   // SR flip-flop
   END_IF;
   IF "Enc"."8BC1.T".refOk THEN #setValueEnc := FALSE; END_IF;
   #T[2].TON(IN := #setValueEnc, PT := t#500ms);
   IF #T[2].Q THEN
       "Enc"."8BC1.T".refOk := TRUE;   // SR flip-flop
   END_IF;
   IF "Enc"."8BC1.T".refRun THEN "Enc"."8BC1.T".refOk := FALSE; END_IF;
END_REGION

REGION Network 14: adj slow - enocder
   IF "G".Cfg.adjTopActive THEN
       #Enc(adr := "Local~-13A1121",   // "SysCounterFast"
            changeDir := false,
            reset := false,
            calOffset := 0.0,
            calGain := "Enc"."8BC1.T".calGain,
            set := NOT "I_8S1.T_in" AND #setValueEnc,
            setValue := "Enc"."8BC1.T".minPos,
            ack := "G".ack,
            runCheckActive := true,
            runCheckTime := T#3s,
            runCheckDiff := 0.01,
            runSig := "Mot"."8M1.T".run,
            errOffDelTime := T#1s,
            limMin := "Enc"."8BC1.T".limMin,
            limMax := "Enc"."8BC1.T".limMax,
            Enc := "Enc"."8BC1.T");
   END_IF;
END_REGION

REGION Network 15: adj slow - pos
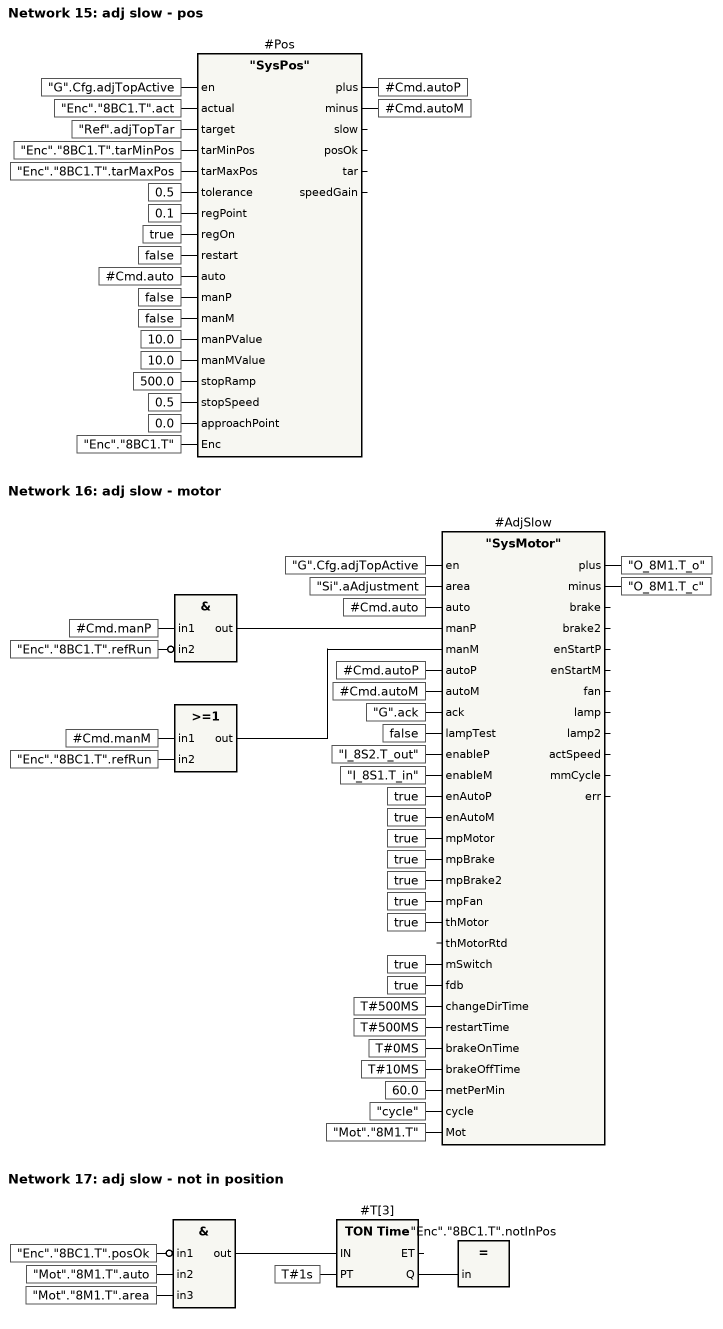
   IF "G".Cfg.adjTopActive THEN
       #Pos(actual := "Enc"."8BC1.T".act,   // "SysPos"
            target := "Ref".adjTopTar,
            tarMinPos := "Enc"."8BC1.T".tarMinPos,
            tarMaxPos := "Enc"."8BC1.T".tarMaxPos,
            tolerance := 0.5,
            regPoint := 0.1,
            regOn := true,
            restart := false,
            auto := #Cmd.auto,
            manP := false,
            manM := false,
            manPValue := 10.0,
            manMValue := 10.0,
            stopRamp := 500.0,
            stopSpeed := 0.5,
            approachPoint := 0.0,
            Enc := "Enc"."8BC1.T",
            plus => #Cmd.autoP,
            minus => #Cmd.autoM);
   END_IF;
END_REGION

REGION Network 16: adj slow - motor
   IF "G".Cfg.adjTopActive THEN
       #AdjSlow(area := "Si".aAdjustment,   // "SysMotor"
                auto := #Cmd.auto,
                manP := #Cmd.manP AND NOT "Enc"."8BC1.T".refRun,
                manM := #Cmd.manM OR "Enc"."8BC1.T".refRun,
                autoP := #Cmd.autoP,
                autoM := #Cmd.autoM,
                ack := "G".ack,
                lampTest := false,
                enableP := "I_8S2.T_out",
                enableM := "I_8S1.T_in",
                enAutoP := true,
                enAutoM := true,
                mpMotor := true,
                mpBrake := true,
                mpBrake2 := true,
                mpFan := true,
                thMotor := true,
                mSwitch := true,
                fdb := true,
                changeDirTime := T#500MS,
                restartTime := T#500MS,
                brakeOnTime := T#0MS,
                brakeOffTime := T#10MS,
                metPerMin := 60.0,
                cycle := "cycle",
                Mot := "Mot"."8M1.T",
                plus => "O_8M1.T_o",
                minus => "O_8M1.T_c");
   END_IF;
END_REGION

REGION Network 17: adj slow - not in position
   #T[3].TON(IN := NOT "Enc"."8BC1.T".posOk AND "Mot"."8M1.T".auto AND "Mot"."8M1.T".area, PT := T#1s);
   "Enc"."8BC1.T".notInPos := #T[3].Q;
END_REGION

REGION Network 18: adj slow - sensor monitoring
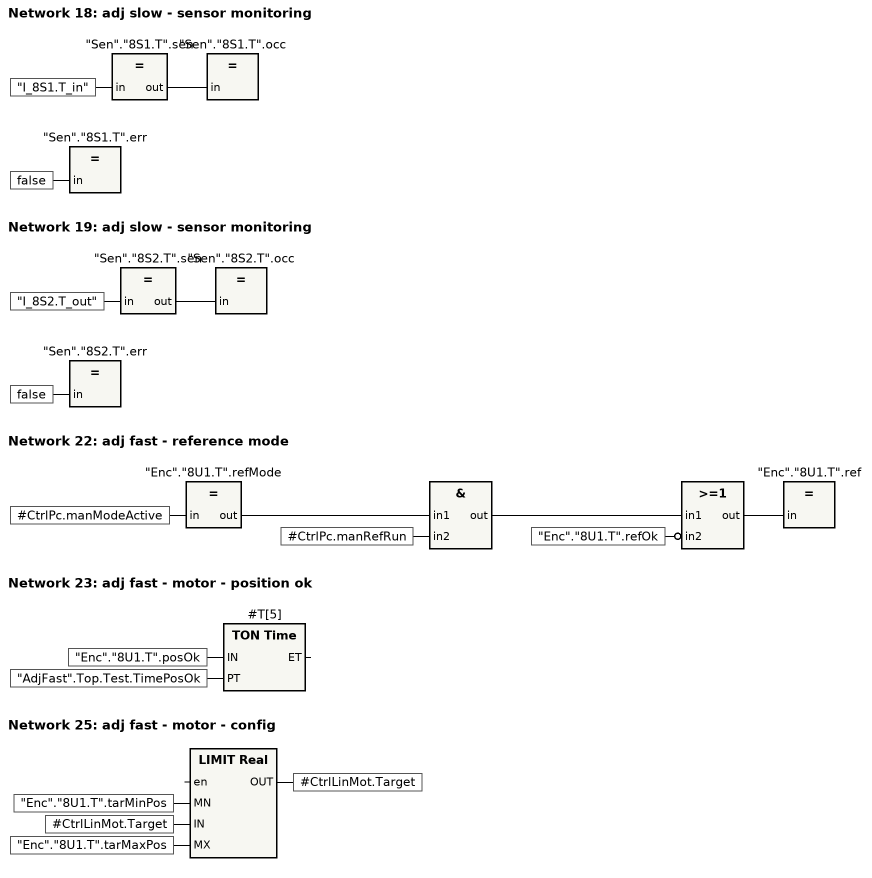
   "Sen"."8S1.T".sen := "I_8S1.T_in";
   "Sen"."8S1.T".occ := "I_8S1.T_in";
   "Sen"."8S1.T".err := false;
END_REGION

REGION Network 19: adj slow - sensor monitoring
   "Sen"."8S2.T".sen := "I_8S2.T_out";
   "Sen"."8S2.T".occ := "I_8S2.T_out";
   "Sen"."8S2.T".err := false;
END_REGION

REGION Network 21 (SCL): adj fast - calibration value
   "Enc"."8U1.T".calGain := 1.0;

   "Enc"."8U1.T".minPos := 5.0;
   "Enc"."8U1.T".maxPos := 155.0;

   "Enc"."8U1.T".limMin := "Enc"."8U1.T".minPos - 5.0;
   "Enc"."8U1.T".limMax := "Enc"."8U1.T".maxPos + 5.0;

   "Enc"."8U1.T".tarMinPos := "Enc"."8U1.T".minPos + 0.0;
   "Enc"."8U1.T".tarMaxPos := "Enc"."8U1.T".maxPos - 0.0;
END_REGION

REGION Network 22: adj fast - reference mode
   "Enc"."8U1.T".refMode := #CtrlPc.manModeActive;
   "Enc"."8U1.T".ref := (#CtrlPc.manModeActive AND #CtrlPc.manRefRun) OR NOT "Enc"."8U1.T".refOk;
END_REGION

REGION Network 23: adj fast - motor - position ok
   #T[5].TON(IN := "Enc"."8U1.T".posOk, PT := "AdjFast".Top.Test.TimePosOk);
END_REGION

REGION Network 24 (SCL): adj fast - motor - config

   //############################################################
   // min            5     mm
   // max          155     mm

   // speed        02      m/s
   // acc/dec      24      m/s2
   // jerk         450     m/s3

   // mode         BestehornVAJ
   //############################################################

   // only testmode for plc
   IF "AdjFast".Top.Test.ModeActive AND NOT #CtrlPc.manModeActive THEN
       IF "AdjFast".Top.Test.TarPos = "AdjFast".Top.Test.TarPos1 AND #T[5].Q THEN
           "AdjFast".Top.Test.TarPos := "AdjFast".Top.Test.TarPos2;
       ELSIF "AdjFast".Top.Test.TarPos = "AdjFast".Top.Test.TarPos2 AND #T[5].Q THEN
           "AdjFast".Top.Test.TarPos := "AdjFast".Top.Test.TarPos1;
       END_IF;
       "Ref".adjTopTar := "AdjFast".Top.Test.TarPos;
   END_IF;

   // active mode
   #CtrlLinMot.Mode := 3;
   #CtrlLinMot.Target := "Ref".adjTopTar;
   #CtrlLinMot.Speed := 2.0;
   #CtrlLinMot.Acc := 24.0;
   #CtrlLinMot.Dec := 0.0;
   #CtrlLinMot.Jerk := 450.0;

   // only testmode for plc
   IF "AdjFast".Top.Mode = 1 THEN
       #CtrlLinMot.Mode := 1;
       #CtrlLinMot.Target := "AdjFast".Top.VAI.Par1;
       #CtrlLinMot.Speed := "AdjFast".Top.VAI.Par2;
       #CtrlLinMot.Acc := "AdjFast".Top.VAI.Par3;
       #CtrlLinMot.Dec := "AdjFast".Top.VAI.Par4;
       #CtrlLinMot.Jerk := 0.0;
   ELSIF "AdjFast".Top.Mode = 2 THEN
       #CtrlLinMot.Mode := 2;
       #CtrlLinMot.Target := "AdjFast".Top.SinVA.Par1;
       #CtrlLinMot.Speed := "AdjFast".Top.SinVA.Par2;
       #CtrlLinMot.Acc := "AdjFast".Top.SinVA.Par3;
       #CtrlLinMot.Dec := 0.0;
       #CtrlLinMot.Jerk := 0.0;
   ELSIF "AdjFast".Top.Mode = 3 THEN
       #CtrlLinMot.Mode := 3;
       #CtrlLinMot.Target := "AdjFast".Top.BestehornVAJ.Par1;
       #CtrlLinMot.Speed := "AdjFast".Top.BestehornVAJ.Par2;
       #CtrlLinMot.Acc := "AdjFast".Top.BestehornVAJ.Par3;
       #CtrlLinMot.Dec := 0.0;
       #CtrlLinMot.Jerk := "AdjFast".Top.BestehornVAJ.Par4;
   END_IF;
END_REGION

REGION Network 25: adj fast - motor - config
   #CtrlLinMot.Target := LIMIT(MN := "Enc"."8U1.T".tarMinPos, IN := #CtrlLinMot.Target, MX := "Enc"."8U1.T".tarMaxPos);
END_REGION

REGION Network 26: adj fast - motor
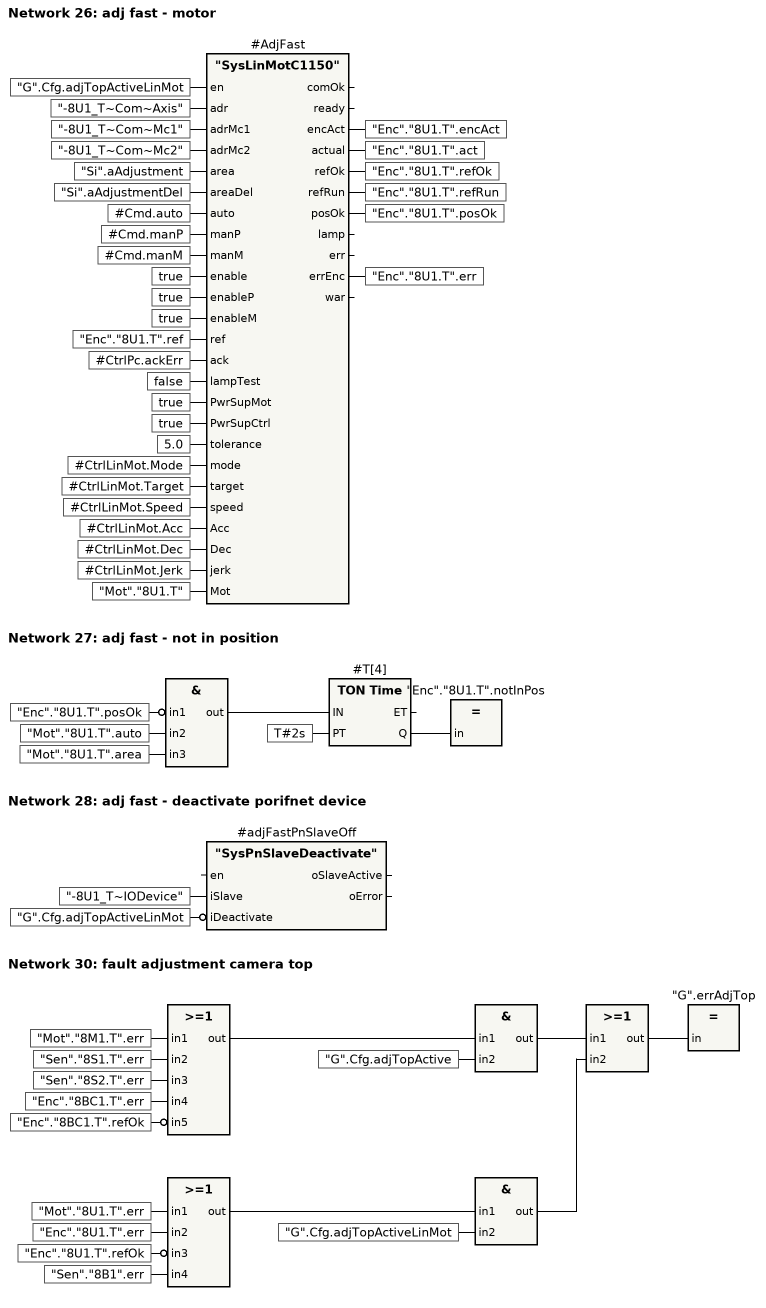
   IF "G".Cfg.adjTopActiveLinMot THEN
       #AdjFast(adr := "-8U1_T~Com~Axis",   // "SysLinMotC1150"
                adrMc1 := "-8U1_T~Com~Mc1",
                adrMc2 := "-8U1_T~Com~Mc2",
                area := "Si".aAdjustment,
                areaDel := "Si".aAdjustmentDel,
                auto := #Cmd.auto,
                manP := #Cmd.manP,
                manM := #Cmd.manM,
                enable := true,
                enableP := true,
                enableM := true,
                ref := "Enc"."8U1.T".ref,
                ack := #CtrlPc.ackErr,
                lampTest := false,
                PwrSupMot := true,
                PwrSupCtrl := true,
                tolerance := 5.0,
                mode := #CtrlLinMot.Mode,
                target := #CtrlLinMot.Target,
                speed := #CtrlLinMot.Speed,
                Acc := #CtrlLinMot.Acc,
                Dec := #CtrlLinMot.Dec,
                jerk := #CtrlLinMot.Jerk,
                Mot := "Mot"."8U1.T",
                encAct => "Enc"."8U1.T".encAct,
                actual => "Enc"."8U1.T".act,
                refOk => "Enc"."8U1.T".refOk,
                refRun => "Enc"."8U1.T".refRun,
                posOk => "Enc"."8U1.T".posOk,
                errEnc => "Enc"."8U1.T".err);
   END_IF;
END_REGION

REGION Network 27: adj fast - not in position
   #T[4].TON(IN := NOT "Enc"."8U1.T".posOk AND "Mot"."8U1.T".auto AND "Mot"."8U1.T".area, PT := T#2s);
   "Enc"."8U1.T".notInPos := #T[4].Q;
END_REGION

REGION Network 28: adj fast - deactivate porifnet device
   #adjFastPnSlaveOff(iSlave := "-8U1_T~IODevice", iDeactivate := NOT "G".Cfg.adjTopActiveLinMot);   // "SysPnSlaveDeactivate"
END_REGION

REGION Network 30: fault adjustment camera top
   "G".errAdjTop := (("Mot"."8M1.T".err OR "Sen"."8S1.T".err OR "Sen"."8S2.T".err OR "Enc"."8BC1.T".err OR NOT "Enc"."8BC1.T".refOk) AND "G".Cfg.adjTopActive) OR (("Mot"."8U1.T".err OR "Enc"."8U1.T".err OR NOT "Enc"."8U1.T".refOk OR "Sen"."8B1".err) AND "G".Cfg.adjTopActiveLinMot);
END_REGION

REGION Network 31 (SCL): data to pc
   IF "G".Cfg.adjTopActive THEN
       "Ref".adjTopAct := REAL_TO_DINT("Enc"."8BC1.T".act * 10.0) - "Ref".adjTopCalOffset - REAL_TO_DINT(#offsetNoStd * 10.0);
       "ComSd".Data.Top.ActualEncPos := REAL_TO_DINT("Enc"."8BC1.T".act * 10.0);
       "ComSd".Data.Top.ActualPos := "Ref".adjTopAct;
       "ComSd".Data.Top.LimitSwitchMin := "Sen"."8S1.T".sen;
       "ComSd".Data.Top.LimitSwitchMax := "Sen"."8S2.T".sen;
       "ComSd".Data.Top.Err := "Mot"."8M1.T".err;
       "ComSd".Data.Top.ErrEnc := "Enc"."8BC1.T".err;
       "ComSd".Data.Top.PosOk := "Enc"."8BC1.T".posOk;
       "ComSd".Data.Top.Plus := "Mot"."8M1.T".plus;
       "ComSd".Data.Top.Minus := "Mot"."8M1.T".minus;
       "ComSd".Data.Top.refRun := "Enc"."8BC1.T".refRun;
       "ComSd".Data.Top.refOk := "Enc"."8BC1.T".refOk;
   ELSIF  "G".Cfg.adjTopActiveLinMot THEN
       "Ref".adjTopAct := REAL_TO_DINT("Enc"."8U1.T".act * 10.0) - "Ref".adjTopCalOffset - REAL_TO_DINT(#offsetNoStd * 10.0);
       "ComSd".Data.Top.ActualEncPos := REAL_TO_DINT("Enc"."8U1.T".act * 10.0);
       "ComSd".Data.Top.ActualPos := "Ref".adjTopAct;
       "ComSd".Data.Top.LimitSwitchMin := TRUE;
       "ComSd".Data.Top.LimitSwitchMax := TRUE;
       "ComSd".Data.Top.Err := "Mot"."8U1.T".err;
       "ComSd".Data.Top.ErrEnc := "Enc"."8U1.T".err;
       "ComSd".Data.Top.PosOk := "Enc"."8U1.T".posOk;
       "ComSd".Data.Top.Plus := "Mot"."8U1.T".plus;
       "ComSd".Data.Top.Minus := "Mot"."8U1.T".minus;
       "ComSd".Data.Top.refRun := "Enc"."8U1.T".refRun;
       "ComSd".Data.Top.refOk := "Enc"."8U1.T".refOk;
   ELSE
       "ComSd".Data.Top.ActualEncPos := 0;
       "ComSd".Data.Top.ActualPos := 0;
       "ComSd".Data.Top.LimitSwitchMin := FALSE;
       "ComSd".Data.Top.LimitSwitchMax := FALSE;
       "ComSd".Data.Top.Err := FALSE;
       "ComSd".Data.Top.ErrEnc := FALSE;
       "ComSd".Data.Top.PosOk := True;
       "ComSd".Data.Top.Plus := FALSE;
       "ComSd".Data.Top.Minus := FALSE;
       "ComSd".Data.Top.refRun := FALSE;
       "ComSd".Data.Top.refOk := TRUE;
   END_IF;
END_REGION

REGION Network 32: current monitoring - auto
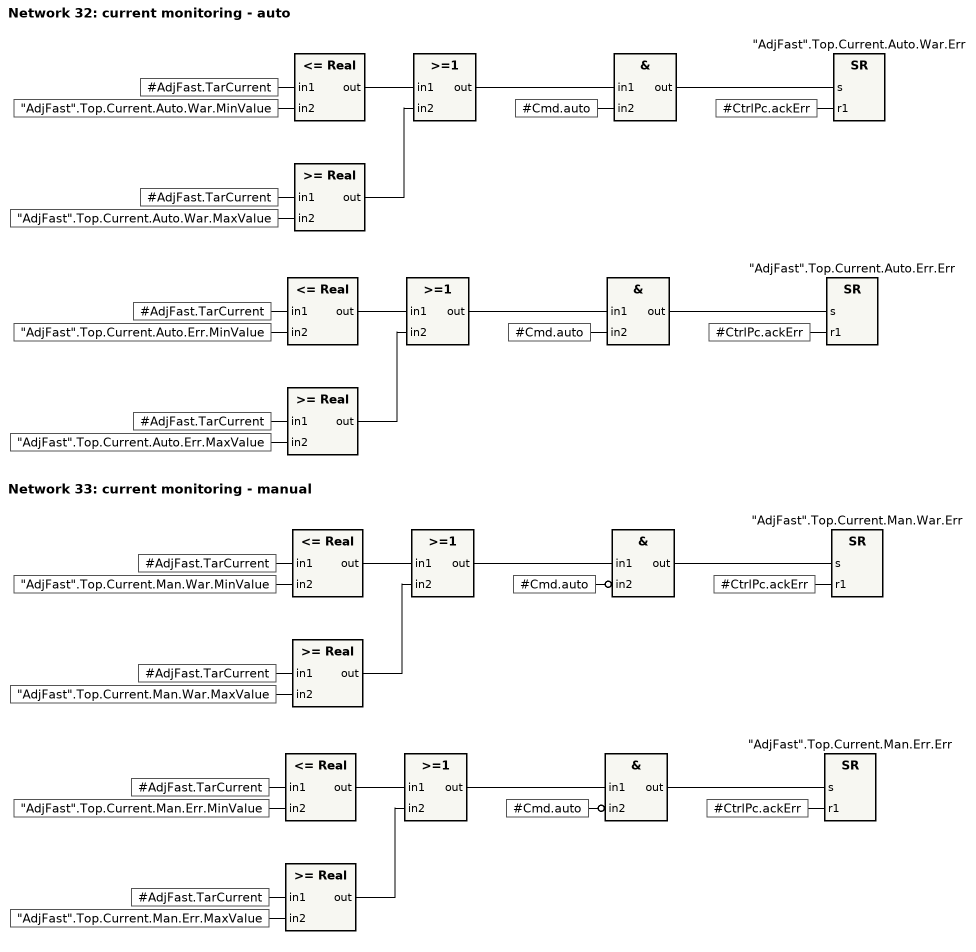
   IF ((#AdjFast.TarCurrent <= "AdjFast".Top.Current.Auto.War.MinValue) OR (#AdjFast.TarCurrent >= "AdjFast".Top.Current.Auto.War.MaxValue)) AND #Cmd.auto THEN
       "AdjFast".Top.Current.Auto.War.Err := TRUE;   // SR flip-flop
   END_IF;
   IF #CtrlPc.ackErr THEN "AdjFast".Top.Current.Auto.War.Err := FALSE; END_IF;
   IF ((#AdjFast.TarCurrent <= "AdjFast".Top.Current.Auto.Err.MinValue) OR (#AdjFast.TarCurrent >= "AdjFast".Top.Current.Auto.Err.MaxValue)) AND #Cmd.auto THEN
       "AdjFast".Top.Current.Auto.Err.Err := TRUE;   // SR flip-flop
   END_IF;
   IF #CtrlPc.ackErr THEN "AdjFast".Top.Current.Auto.Err.Err := FALSE; END_IF;
END_REGION

REGION Network 33: current monitoring - manual
   IF ((#AdjFast.TarCurrent <= "AdjFast".Top.Current.Man.War.MinValue) OR (#AdjFast.TarCurrent >= "AdjFast".Top.Current.Man.War.MaxValue)) AND NOT #Cmd.auto THEN
       "AdjFast".Top.Current.Man.War.Err := TRUE;   // SR flip-flop
   END_IF;
   IF #CtrlPc.ackErr THEN "AdjFast".Top.Current.Man.War.Err := FALSE; END_IF;
   IF ((#AdjFast.TarCurrent <= "AdjFast".Top.Current.Man.Err.MinValue) OR (#AdjFast.TarCurrent >= "AdjFast".Top.Current.Man.Err.MaxValue)) AND NOT #Cmd.auto THEN
       "AdjFast".Top.Current.Man.Err.Err := TRUE;   // SR flip-flop
   END_IF;
   IF #CtrlPc.ackErr THEN "AdjFast".Top.Current.Man.Err.Err := FALSE; END_IF;
END_REGION
END_FUNCTION_BLOCK

FUNCTION_BLOCK "SysLinMotC1150"   // FB2080, FBD
TITLE = manage the positioning over the "extended bus positioning" [6Word]
{ S7_Optimized_Access := 'TRUE' }
AUTHOR : MiCROTEC
VERSION : 1.6
// -2019.12 : Martin
// stored: AutoNumber false, MemoryReserve 100, SetENOAutomatically false
   VAR_INPUT
      adr { ExternalAccessible := 'False'; ExternalVisible := 'False'; ExternalWritable := 'False'} : HW_IO;   // I/O address
      adrMc1 { ExternalAccessible := 'False'; ExternalVisible := 'False'; ExternalWritable := 'False'} : HW_IO;   // I/O address monitoring channel 1
      adrMc2 { ExternalAccessible := 'False'; ExternalVisible := 'False'; ExternalWritable := 'False'} : HW_IO;   // I/O address monitoring channel 2
      area { ExternalAccessible := 'False'; ExternalVisible := 'False'; ExternalWritable := 'False'} : Bool;   // 1=Safety area on
      areaDel { ExternalAccessible := 'False'; ExternalVisible := 'False'; ExternalWritable := 'False'} : Bool;   // 1=safety area on off-delayed
      auto { ExternalAccessible := 'False'; ExternalVisible := 'False'; ExternalWritable := 'False'} : Bool;   // automatic
      manP { ExternalAccessible := 'False'; ExternalVisible := 'False'; ExternalWritable := 'False'} : Bool;   // manual plus
      manM { ExternalAccessible := 'False'; ExternalVisible := 'False'; ExternalWritable := 'False'} : Bool;   // manual minus
      enable { ExternalAccessible := 'False'; ExternalVisible := 'False'; ExternalWritable := 'False'} : Bool;   // enable positioning
      enableP { ExternalAccessible := 'False'; ExternalVisible := 'False'; ExternalWritable := 'False'} : Bool;   // release plus
      enableM { ExternalAccessible := 'False'; ExternalVisible := 'False'; ExternalWritable := 'False'} : Bool;   // release minus
      ref { ExternalAccessible := 'False'; ExternalVisible := 'False'; ExternalWritable := 'False'} : Bool;   // reference
      ack { ExternalAccessible := 'False'; ExternalVisible := 'False'; ExternalWritable := 'False'} : Bool;   // fault acknowledge
      lampTest { ExternalAccessible := 'False'; ExternalVisible := 'False'; ExternalWritable := 'False'} : Bool;   // lamptest
      PwrSupMot { ExternalAccessible := 'False'; ExternalVisible := 'False'; ExternalWritable := 'False'} : Bool;   // 1=power supply motor ok / 1=motor protection switch ok
      PwrSupCtrl { ExternalAccessible := 'False'; ExternalVisible := 'False'; ExternalWritable := 'False'} : Bool;   // 1=power supply controller ok / 1=Motor protection switch brake ok
      tolerance { ExternalAccessible := 'False'; ExternalVisible := 'False'; ExternalWritable := 'False'} : Real;   // tolerance for output signal position ok
      mode { ExternalAccessible := 'False'; ExternalVisible := 'False'; ExternalWritable := 'False'} : Int;   // 1=VAI / 2=SIN VA / 3=Bestehorn VAJ
      target { ExternalAccessible := 'False'; ExternalVisible := 'False'; ExternalWritable := 'False'} : Real;   // target position [mm] / target position
      speed { ExternalAccessible := 'False'; ExternalVisible := 'False'; ExternalWritable := 'False'} : Real;   // target speed [m/s ] / target speed [ 1/min ]
      Acc { ExternalAccessible := 'False'; ExternalVisible := 'False'; ExternalWritable := 'False'} : Real;   // acceleration [m/s2] / start ramp [ms]
      Dec { ExternalAccessible := 'False'; ExternalVisible := 'False'; ExternalWritable := 'False'} : Real;   // deceleration [m/s2] / stop ramp [ms]
      jerk { ExternalAccessible := 'False'; ExternalVisible := 'False'; ExternalWritable := 'False'} : Real;   // jerk [m/s3]
   END_VAR
   VAR_OUTPUT
      comOk { ExternalAccessible := 'False'; ExternalVisible := 'False'; ExternalWritable := 'False'} : Bool;   // frequency converter communication ok
      ready { ExternalAccessible := 'False'; ExternalVisible := 'False'; ExternalWritable := 'False'} : Bool;   // frequency converter ready
      encAct { ExternalAccessible := 'False'; ExternalVisible := 'False'; ExternalWritable := 'False'} : DInt;   // actual position [inc]
      actual { ExternalAccessible := 'False'; ExternalVisible := 'False'; ExternalWritable := 'False'} : Real;   // actual position
      refOk { ExternalAccessible := 'False'; ExternalVisible := 'False'; ExternalWritable := 'False'} : Bool;   // reference ok
      refRun { ExternalAccessible := 'False'; ExternalVisible := 'False'; ExternalWritable := 'False'} : Bool;   // reference run active
      posOk { ExternalAccessible := 'False'; ExternalVisible := 'False'; ExternalWritable := 'False'} : Bool;   // position ok
      lamp { ExternalAccessible := 'False'; ExternalVisible := 'False'; ExternalWritable := 'False'} : Bool;   // indication lamp
      err { ExternalAccessible := 'False'; ExternalVisible := 'False'; ExternalWritable := 'False'} : Bool;   // fault
      errEnc { ExternalAccessible := 'False'; ExternalVisible := 'False'; ExternalWritable := 'False'} : Bool;   // fault encoder
      war { ExternalAccessible := 'False'; ExternalVisible := 'False'; ExternalWritable := 'False'} : Bool;   // warning
   END_VAR
   VAR_IN_OUT
      Mot : "TypeMotor";   // data motor
   END_VAR
   VAR
      var { ExternalAccessible := 'False'; ExternalVisible := 'False'; ExternalWritable := 'False'} : Struct
         "bool" : Bool;
         "byte" : Byte;
         "word" : Word;
         "dword" : DWord;
         "int" : Int;
         "dint" : DInt;
         "real" : Real;
         s5time : S5Time;
         "time" : Time;
         hm : Array[1..16] of Bool;
         fm : Array[1..16] of Bool;
      END_STRUCT;
      Rd { ExternalAccessible := 'False'; ExternalVisible := 'False'; ExternalWritable := 'False'} : "TypeLinmotRd";
      RdMc1 { ExternalAccessible := 'False'; ExternalVisible := 'False'; ExternalWritable := 'False'} : DInt;   // actual velocity
      RdMc2 { ExternalAccessible := 'False'; ExternalVisible := 'False'; ExternalWritable := 'False'} : DInt;   // actual error code
      Sd { ExternalAccessible := 'False'; ExternalVisible := 'False'; ExternalWritable := 'False'} : "TypeLinmotSd";
      T { ExternalAccessible := 'False'; ExternalVisible := 'False'; ExternalWritable := 'False'} : Array[1..8] of IEC_TIMER;
      errNrOld { ExternalAccessible := 'False'; ExternalVisible := 'False'; ExternalWritable := 'False'} : UDInt;
      man { ExternalAccessible := 'False'; ExternalVisible := 'False'; ExternalWritable := 'False'} : Bool;
      autoOld { ExternalAccessible := 'False'; ExternalVisible := 'False'; ExternalWritable := 'False'} : Bool;
      errGen { ExternalAccessible := 'False'; ExternalVisible := 'False'; ExternalWritable := 'False'} : Bool;
      enOnDel { ExternalAccessible := 'False'; ExternalVisible := 'False'; ExternalWritable := 'False'} : Bool;
      MotEnable { ExternalAccessible := 'False'; ExternalVisible := 'False'; ExternalWritable := 'False'} : Bool;
      MotSwitchOn { ExternalAccessible := 'False'; ExternalVisible := 'False'; ExternalWritable := 'False'} : Bool;
      statReady { ExternalAccessible := 'False'; ExternalVisible := 'False'; ExternalWritable := 'False'} : Bool;
      statCtrlAuto { ExternalAccessible := 'False'; ExternalVisible := 'False'; ExternalWritable := 'False'} : Bool;
      TarPos { ExternalAccessible := 'False'; ExternalVisible := 'False'; ExternalWritable := 'False'} : Real;
      TarCurrent { ExternalAccessible := 'False'; ExternalVisible := 'False'; ExternalWritable := 'False'} : Real;
      TimeResetHome { ExternalAccessible := 'False'; ExternalVisible := 'False'; ExternalWritable := 'False'} : TON_TIME;
      targetOld { ExternalAccessible := 'False'; ExternalVisible := 'False'; ExternalWritable := 'False'} : Real;
      StartPos { ExternalAccessible := 'False'; ExternalVisible := 'False'; ExternalWritable := 'False'} : Bool;
      PosTolOk { ExternalAccessible := 'False'; ExternalVisible := 'False'; ExternalWritable := 'False'} : Bool;
      TimeStartPos { ExternalAccessible := 'False'; ExternalVisible := 'False'; ExternalWritable := 'False'} : TP_TIME;
      McPar4 { ExternalAccessible := 'False'; ExternalVisible := 'False'; ExternalWritable := 'False'} : Real;
      Mc1 { ExternalAccessible := 'False'; ExternalVisible := 'False'; ExternalWritable := 'False'} : DInt;
      Mc2 { ExternalAccessible := 'False'; ExternalVisible := 'False'; ExternalWritable := 'False'} : DInt;
   END_VAR
   VAR_TEMP
      tempSdRetVal : Int;
      tempRdRetVal1 : Int;
      tempRdRetVal2 : Int;
      tempRdRetVal3 : Int;
      tempName : WString[20];
      tempDescription : WString[60];
      label : WString[26];
      tempString : WString;
      tempStrgPointer : Int;
      tempAck : Bool;
      tempStat : Bool;
      tempWar : Bool;
      tempOp : DInt;
      tempRd : Array[0..3] of Byte;
      tempDint : DInt;
      tempSd : Array[0..3] of Byte;
   END_VAR
   VAR_TEMP   // added for the SCL form of the ladder/FBD networks
      _w1 : Bool;
      _w2 : Bool;
   END_VAR
BEGIN

REGION Network 1 (SCL): description
   // Linmot  PL01-20x800/740-HP  Motor Stange Noale
   // control of a linmot motor
   // controller:  Linmot C1150-PN-XC-1S
   // stator:      Linmot PS01-37Sx120F-HP-N-AGI
   // stroke:      Linmot PL01-20x360/300-HP
   // creator:     Alexander Kiebacher
   // version:     1.0
   //
END_REGION

REGION Network 2: exit
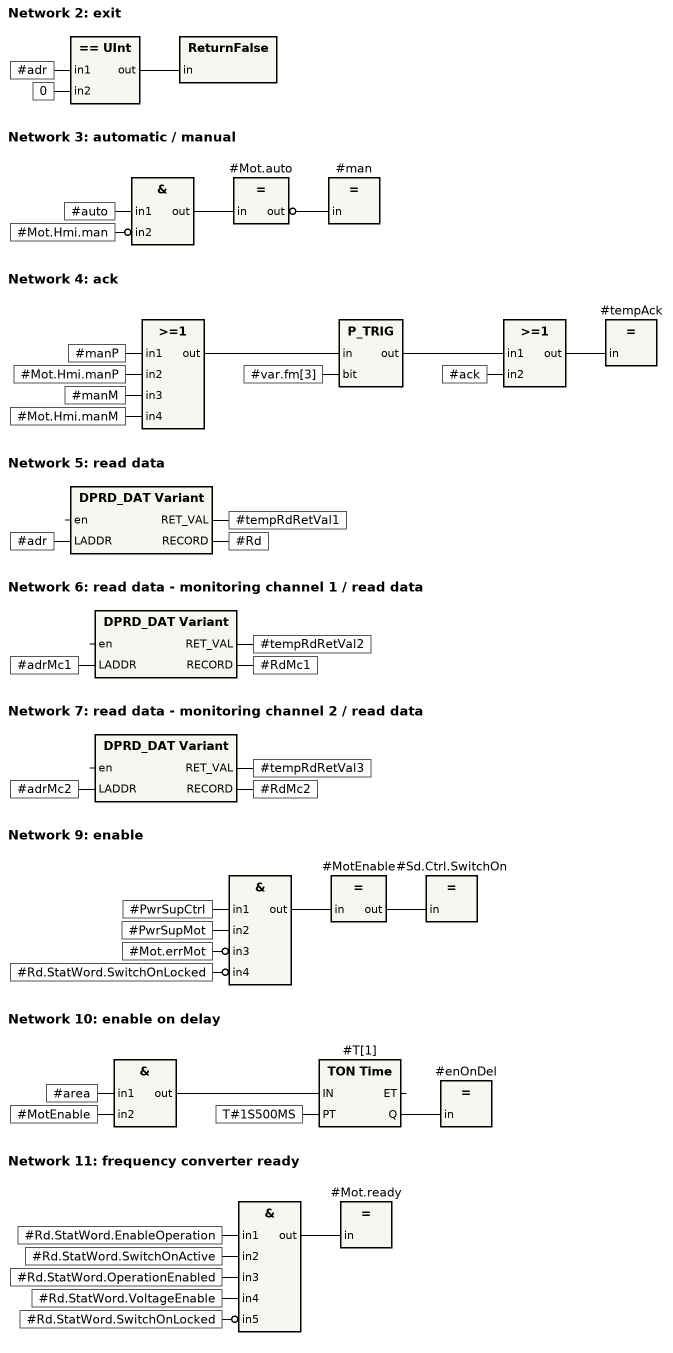
   IF #adr = 0 THEN
       ENO := FALSE;
       RETURN;
   END_IF;
END_REGION

REGION Network 3: automatic / manual
   #_w1 := #auto AND NOT #Mot.Hmi.man;
   #Mot.auto := #_w1;
   #man := NOT #_w1;
END_REGION

REGION Network 4: ack
   #_w1 := #manP OR #Mot.Hmi.manP OR #manM OR #Mot.Hmi.manM;
   #_w2 := #_w1 AND NOT #var.fm[3];   // rising edge
   #var.fm[3] := #_w1;
   #tempAck := #_w2 OR #ack;
END_REGION

REGION Network 5: read data
   #tempRdRetVal1 := DPRD_DAT(LADDR := #adr, RECORD => #Rd);
END_REGION

REGION Network 6: read data - monitoring channel 1 / read data
   #tempRdRetVal2 := DPRD_DAT(LADDR := #adrMc1, RECORD => #RdMc1);
END_REGION

REGION Network 7: read data - monitoring channel 2 / read data
   #tempRdRetVal3 := DPRD_DAT(LADDR := #adrMc2, RECORD => #RdMc2);
END_REGION

REGION Network 8 (SCL): read

   // actual position
   #tempRd[0] := #Rd.Actpos.%B0;
   #tempRd[1] := #Rd.Actpos.%B1;
   #tempRd[2] := #Rd.Actpos.%B2;
   #tempRd[3] := #Rd.Actpos.%B3;

   #Rd.Actpos.%B0 := #tempRd[3];
   #Rd.Actpos.%B1 := #tempRd[2];
   #Rd.Actpos.%B2 := #tempRd[1];
   #Rd.Actpos.%B3 := #tempRd[0];

   #encAct := #Rd.Actpos;
   #actual := DINT_TO_REAL(#Rd.Actpos) / 10000.0;

   // target position
   #tempRd[0] := #Rd.Tarpos.%B0;
   #tempRd[1] := #Rd.Tarpos.%B1;
   #tempRd[2] := #Rd.Tarpos.%B2;
   #tempRd[3] := #Rd.Tarpos.%B3;

   #Rd.Tarpos.%B0 := #tempRd[3];
   #Rd.Tarpos.%B1 := #tempRd[2];
   #Rd.Tarpos.%B2 := #tempRd[1];
   #Rd.Tarpos.%B3 := #tempRd[0];

   #TarPos := DINT_TO_REAL(#Rd.Tarpos) / 10000.0;

   // target current
   #tempRd[0] := #Rd.TarCurrent.%B0;
   #tempRd[1] := #Rd.TarCurrent.%B1;
   #tempRd[2] := #Rd.TarCurrent.%B2;
   #tempRd[3] := #Rd.TarCurrent.%B3;

   #Rd.TarCurrent.%B0 := #tempRd[3];
   #Rd.TarCurrent.%B1 := #tempRd[2];
   #Rd.TarCurrent.%B2 := #tempRd[1];
   #Rd.TarCurrent.%B3 := #tempRd[0];

   #TarCurrent := DINT_TO_REAL(#Rd.TarCurrent) / 1000.0;

   // monitoring channel 1 - target velocity [1000*m/s]
   #tempRd[0] := #RdMc1.%B0;
   #tempRd[1] := #RdMc1.%B1;
   #tempRd[2] := #RdMc1.%B2;
   #tempRd[3] := #RdMc1.%B3;

   #RdMc1.%B0 := #tempRd[3];
   #RdMc1.%B1 := #tempRd[2];
   #RdMc1.%B2 := #tempRd[1];
   #RdMc1.%B3 := #tempRd[0];

   #Mc1 := #RdMc1;

   IF #Rd.StatWord.MotionActive THEN
       IF #Mc1 >= 100 THEN
           #Mot.speedAct := DINT_TO_INT(#Mc1/1000);
       ELSIF #Mc1 <= -100 THEN
           #Mot.speedAct := DINT_TO_INT(#Mc1/1000);
       END_IF;
   ELSE
       #Mot.speedAct := 0;
   END_IF;

   // monitoring channel 2 - actual error code
   #tempRd[0] := #RdMc2.%B0;
   #tempRd[1] := #RdMc2.%B1;
   #tempRd[2] := #RdMc2.%B2;
   #tempRd[3] := #RdMc2.%B3;

   #RdMc2.%B0 := #tempRd[3];
   #RdMc2.%B1 := #tempRd[2];
   #RdMc2.%B2 := #tempRd[1];
   #RdMc2.%B3 := #tempRd[0];

   #Mc2 := #RdMc2;
END_REGION

REGION Network 9: enable
   #MotEnable := #PwrSupCtrl AND #PwrSupMot AND NOT #Mot.errMot AND NOT #Rd.StatWord.SwitchOnLocked;
   #Sd.Ctrl.SwitchOn := #MotEnable;
END_REGION

REGION Network 10: enable on delay
   #T[1].TON(IN := #area AND #MotEnable, PT := T#1S500MS);
   #enOnDel := #T[1].Q;
END_REGION

REGION Network 11: frequency converter ready
   #Mot.ready := #Rd.StatWord.EnableOperation AND #Rd.StatWord.SwitchOnActive AND #Rd.StatWord.OperationEnabled AND #Rd.StatWord.VoltageEnable AND NOT #Rd.StatWord.SwitchOnLocked;
END_REGION

REGION Network 12: ready
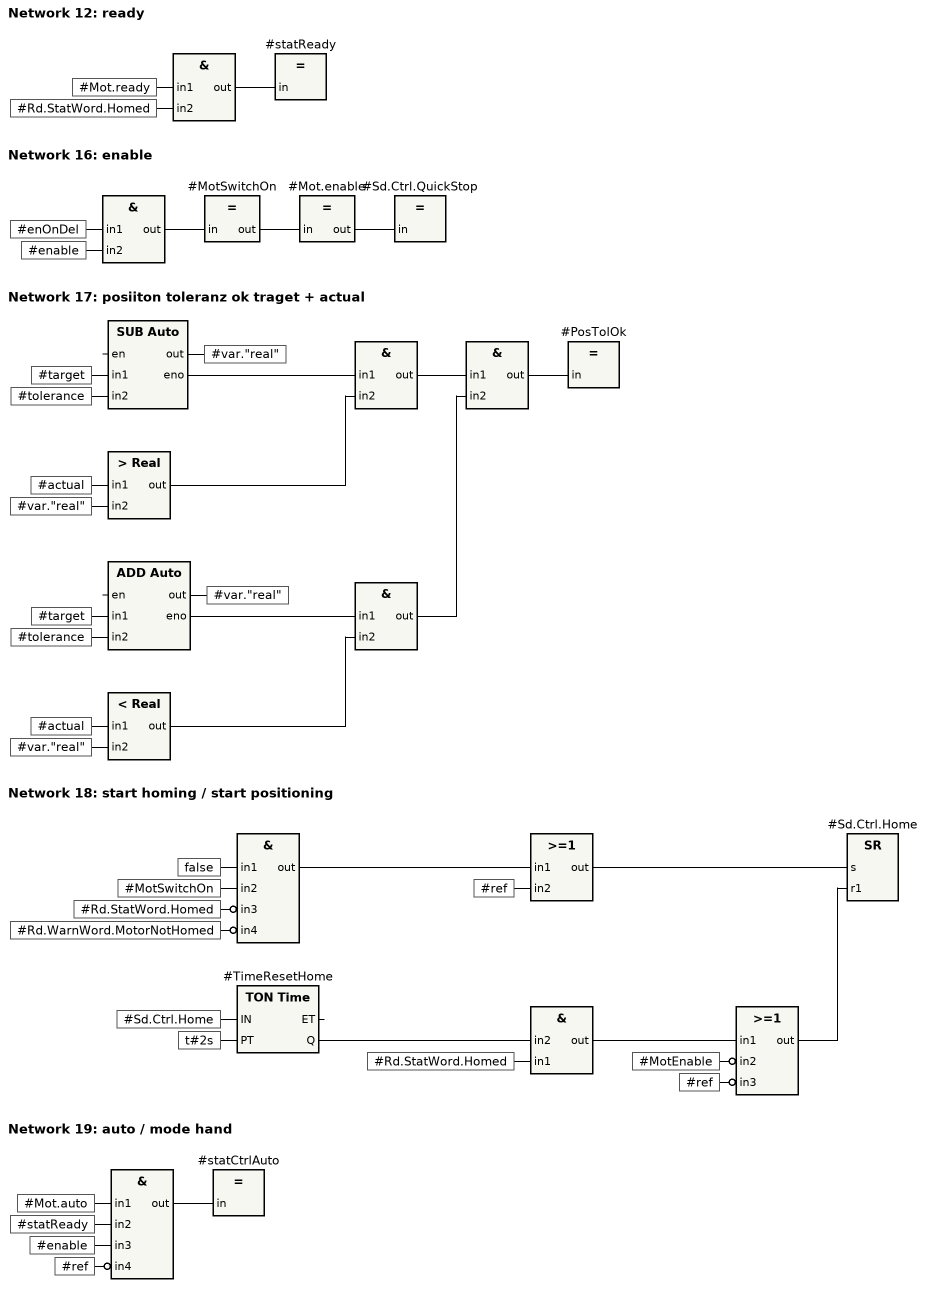
   #statReady := #Mot.ready AND #Rd.StatWord.Homed;
END_REGION

NETWORK
TITLE = test status var

      L     #Rd.StatVar.MainState;  // Op. Main State
      L     #Rd.StatVar.SubState;  // Op. Sub State

      T     #tempOp;


NETWORK
TITLE = test status word

// not used
      O     #Rd.StatWord.EventHandlerActive;
      O     #Rd.StatWord.SpecialMotionActive;
      O     #Rd.StatWord.MotionActive;
      O     #Rd.StatWord.RangeIndicator1;
      O     #Rd.StatWord.RangeIndicator2;
      =     #tempStat;


NETWORK
TITLE = test warning word

// not used
      O     #Rd.StatWord.Warning;
      O     #Rd.WarnWord.MotorHotSensor;
      O     #Rd.WarnWord.MotorShortTimerOverload;
      O     #Rd.WarnWord.MotorSupplyVoltageLow;
      O     #Rd.WarnWord.MotorSupplyVoltageHigh;
      O     #Rd.WarnWord.PositionLagAlways;
      O     #Rd.WarnWord.Res5;
      O     #Rd.WarnWord.DriveHot;
      O     #Rd.WarnWord.PTC_Sensor1Hot;
      O     #Rd.WarnWord.PTC_Sensor2Hot;
      O     #Rd.WarnWord.Res10;
      O     #Rd.WarnWord.Res11;
      O     #Rd.WarnWord.Res12;
      O     #Rd.WarnWord.Res13;
      O     #Rd.WarnWord.InterfaceWarnFlag;
      O     #Rd.WarnWord.ApplicationWarnFlag;
      =     #tempWar;


REGION Network 16: enable
   #MotSwitchOn := #enOnDel AND #enable;
   #Mot.enable := #MotSwitchOn;
   #Sd.Ctrl.QuickStop := #MotSwitchOn;
END_REGION

REGION Network 17: posiiton toleranz ok traget + actual
   #var."real" := #target - #tolerance;
   #_w1 := #actual > #var."real";
   #var."real" := #target + #tolerance;
   #PosTolOk := #_w1 AND (#actual < #var."real");
END_REGION

REGION Network 18: start homing / start positioning
   // auto reference?
   #TimeResetHome(IN := #Sd.Ctrl.Home, PT := t#2s);   // TON
   IF (false AND #MotSwitchOn AND NOT #Rd.StatWord.Homed AND NOT #Rd.WarnWord.MotorNotHomed) OR #ref THEN
       #Sd.Ctrl.Home := TRUE;   // SR flip-flop
   END_IF;
   IF (#TimeResetHome.Q AND #Rd.StatWord.Homed) OR NOT #MotEnable OR NOT #ref THEN
       #Sd.Ctrl.Home := FALSE;
   END_IF;
END_REGION

REGION Network 19: auto / mode hand
   #statCtrlAuto := #Mot.auto AND #statReady AND #enable AND NOT #ref;
END_REGION

REGION Network 20: start positioning
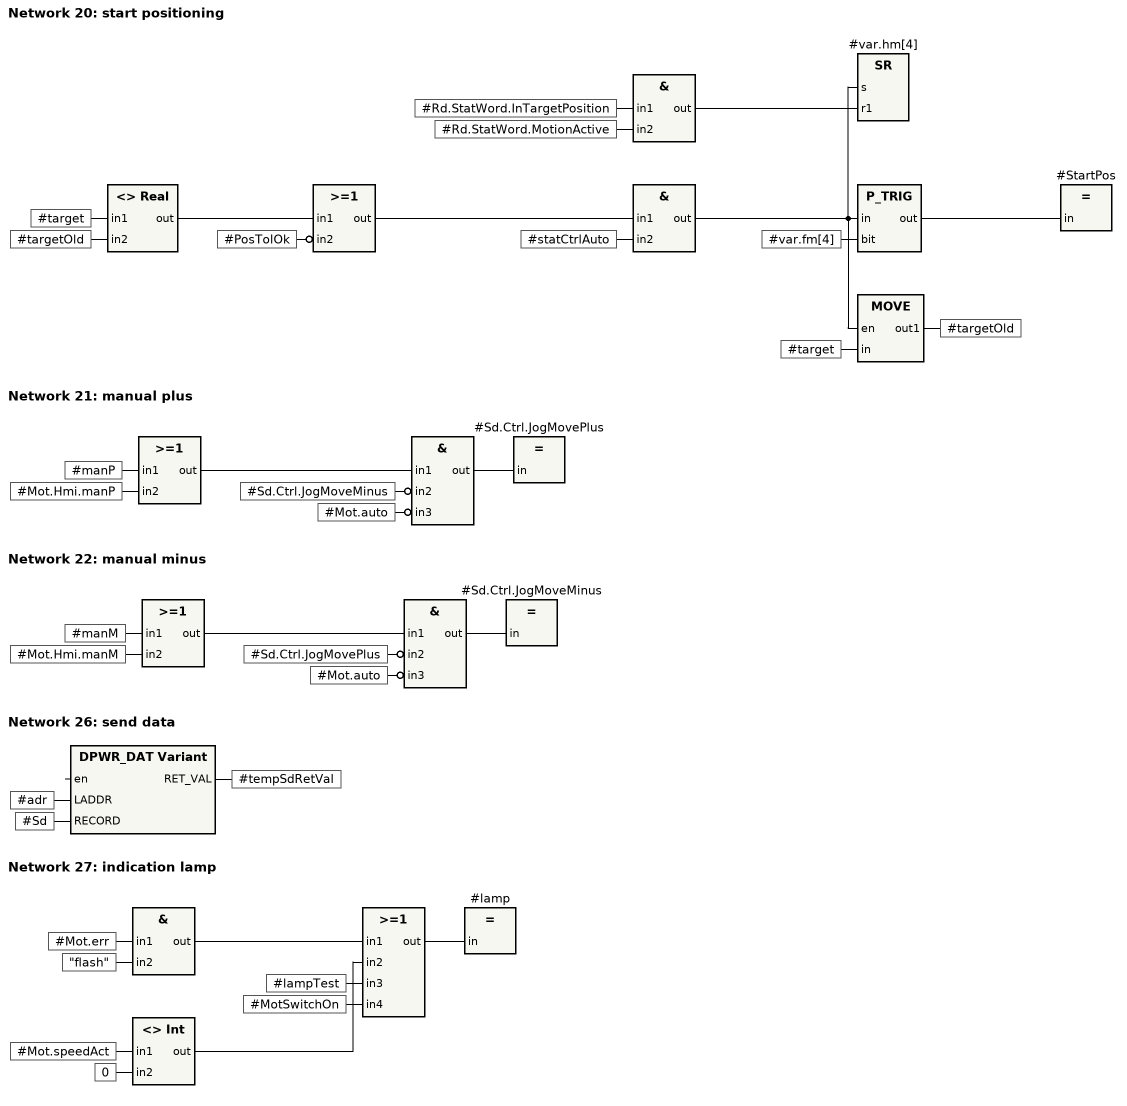
   #_w1 := ((#target <> #targetOld) OR NOT #PosTolOk) AND #statCtrlAuto;
   IF #_w1 THEN
       #var.hm[4] := TRUE;   // SR flip-flop
   END_IF;
   IF #Rd.StatWord.InTargetPosition AND #Rd.StatWord.MotionActive THEN #var.hm[4] := FALSE; END_IF;
   #_w2 := #_w1 AND NOT #var.fm[4];   // rising edge
   #var.fm[4] := #_w1;
   #StartPos := #_w2;
   IF #_w1 THEN #targetOld := #target; END_IF;
END_REGION

REGION Network 21: manual plus
   #Sd.Ctrl.JogMovePlus := (#manP OR #Mot.Hmi.manP) AND NOT #Sd.Ctrl.JogMoveMinus AND NOT #Mot.auto;
END_REGION

REGION Network 22: manual minus
   #Sd.Ctrl.JogMoveMinus := (#manM OR #Mot.Hmi.manM) AND NOT #Sd.Ctrl.JogMovePlus AND NOT #Mot.auto;
END_REGION

REGION Network 23 (SCL)

   #Sd.Ctrl.EnableOperation := TRUE;          // Forced
   #Sd.Ctrl.Abort := TRUE;                    // Forced
   #Sd.Ctrl.Freeze := TRUE;                   // Forced

   // not used
   #Sd.Ctrl.VoltageEnable := FALSE;            // STO
   #Sd.Ctrl.GoToPosition := FALSE;
   #Sd.Ctrl.SpecialMove := FALSE;
   #Sd.Ctrl.ClearanceCheck := FALSE;
   #Sd.Ctrl.GoToInitialPosition := FALSE;
   #Sd.Ctrl.Linearizing := FALSE;
   #Sd.Ctrl.PhaseSearch := FALSE;
END_REGION

REGION Network 24 (SCL): write - MC Header / write

   // Command Count
   // A new command will only be executed, if the value of the command count has changed. In the easiest way bit 0 can be toggled
   #Sd.McHd.CC0 := #StartPos;
   #Sd.McHd.CC1 := FALSE;
   #Sd.McHd.CC2 := FALSE;
   #Sd.McHd.CC3 := FALSE;

   // Master ID
   #Sd.McHd.MasterID := B#16#00;
   IF #mode = 1 THEN
       // VAI
       #Sd.McHd.MasterID := B#16#01;
   ELSIF #mode = 2 THEN
       // SIN VA
       #Sd.McHd.MasterID := B#16#0E;
   ELSIF #mode = 3 THEN
       // Bestehorn VAJ
       #Sd.McHd.MasterID := B#16#0F;
   END_IF;

   // not used Sub ID
   #Sd.McHd.SubID0 := FALSE;
   #Sd.McHd.SubID1 := FALSE;
   #Sd.McHd.SubID2 := FALSE;
   #Sd.McHd.SubID3 := FALSE;
END_REGION

REGION Network 25 (SCL): write - MC Parameter / write

   #Sd.McPar1 := L#0;
   #Sd.McPar2 := L#0;
   #Sd.McPar3 := L#0;
   #Sd.McPar4 := L#0;

   // McPar1 - target
   // 
   #tempDint := REAL_TO_DINT(#target * 10000.0);
   #tempSd[0] := #tempDint.%B0;
   #tempSd[1] := #tempDint.%B1;
   #tempSd[2] := #tempDint.%B2;
   #tempSd[3] := #tempDint.%B3;

   #Sd.McPar1.%B0 := #tempSd[3];
   #Sd.McPar1.%B1 := #tempSd[2];
   #Sd.McPar1.%B2 := #tempSd[1];
   #Sd.McPar1.%B3 := #tempSd[0];

   // McPar2 - speed
   // 
   #tempDint := REAL_TO_DINT(#speed * 1000000.0);
   #tempSd[0] := #tempDint.%B0;
   #tempSd[1] := #tempDint.%B1;
   #tempSd[2] := #tempDint.%B2;
   #tempSd[3] := #tempDint.%B3;

   #Sd.McPar2.%B0 := #tempSd[3];
   #Sd.McPar2.%B1 := #tempSd[2];
   #Sd.McPar2.%B2 := #tempSd[1];
   #Sd.McPar2.%B3 := #tempSd[0];

   // McPar3
   // VAI              - acc
   // SIN VA           - acc/dec
   // Bestehorn VAJ    - acc/dec
   #tempDint := REAL_TO_DINT(#Acc * 100000.0);
   #tempSd[0] := #tempDint.%B0;
   #tempSd[1] := #tempDint.%B1;
   #tempSd[2] := #tempDint.%B2;
   #tempSd[3] := #tempDint.%B3;

   #Sd.McPar3.%B0 := #tempSd[3];
   #Sd.McPar3.%B1 := #tempSd[2];
   #Sd.McPar3.%B2 := #tempSd[1];
   #Sd.McPar3.%B3 := #tempSd[0];

   // McPar4
   #McPar4 := 0.0;
   #tempDint := 0;
   IF #mode = 1 THEN
       // VAI
       #McPar4 := #Dec;
       #tempDint := REAL_TO_DINT(#McPar4 * 100000.0);
   ELSIF #mode = 2 THEN
       // SIN VA
       #McPar4 := 0.0;
       #tempDint := REAL_TO_DINT(#McPar4 * 100000.0);
   ELSIF #mode = 3 THEN
       // Bestehorn VAJ
       #McPar4 := #jerk;
       #tempDint := REAL_TO_DINT(#McPar4 * 10000.0);
   END_IF;

   #tempSd[0] := #tempDint.%B0;
   #tempSd[1] := #tempDint.%B1;
   #tempSd[2] := #tempDint.%B2;
   #tempSd[3] := #tempDint.%B3;

   #Sd.McPar4.%B0 := #tempSd[3];
   #Sd.McPar4.%B1 := #tempSd[2];
   #Sd.McPar4.%B2 := #tempSd[1];
   #Sd.McPar4.%B3 := #tempSd[0];
END_REGION

REGION Network 26: send data
   #tempSdRetVal := DPWR_DAT(LADDR := #adr, RECORD := #Sd);
END_REGION

REGION Network 27: indication lamp
   #lamp := (#Mot.err AND "flash") OR (#Mot.speedAct <> 0) OR #lampTest OR #MotSwitchOn;
END_REGION

REGION Network 28: communication ok
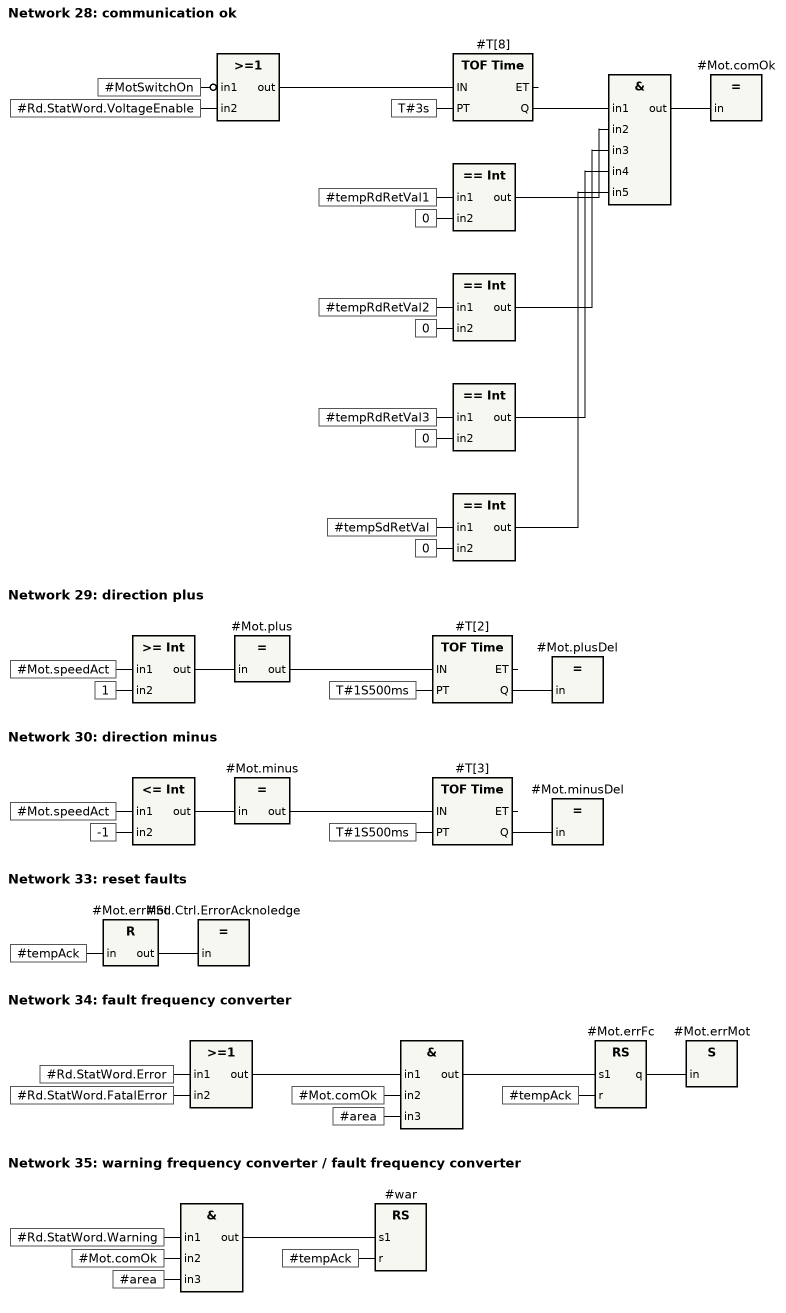
   #T[8].TOF(IN := NOT #MotSwitchOn OR #Rd.StatWord.VoltageEnable, PT := T#3s);
   #Mot.comOk := #T[8].Q AND (#tempRdRetVal1 = 0) AND (#tempRdRetVal2 = 0) AND (#tempRdRetVal3 = 0) AND (#tempSdRetVal = 0);
END_REGION

REGION Network 29: direction plus
   #Mot.plus := #Mot.speedAct >= 1;
   #T[2].TOF(IN := #Mot.plus, PT := T#1S500ms);
   #Mot.plusDel := #T[2].Q;
END_REGION

REGION Network 30: direction minus
   #Mot.minus := #Mot.speedAct <= (-1);
   #T[3].TOF(IN := #Mot.minus, PT := T#1S500ms);
   #Mot.minusDel := #T[3].Q;
END_REGION

REGION Network 32: --faults--
END_REGION

REGION Network 33: reset faults
   IF #tempAck THEN #Mot.errMot := FALSE; END_IF;
   #Sd.Ctrl.ErrorAcknoledge := #tempAck;
END_REGION

REGION Network 34: fault frequency converter
   IF #tempAck THEN
       #Mot.errFc := FALSE;   // RS flip-flop
   END_IF;
   IF (#Rd.StatWord.Error OR #Rd.StatWord.FatalError) AND #Mot.comOk AND #area THEN
       #Mot.errFc := TRUE;
   END_IF;
   IF #Mot.errFc THEN #Mot.errMot := TRUE; END_IF;
END_REGION

REGION Network 35: warning frequency converter / fault frequency converter
   IF #tempAck THEN
       #war := FALSE;   // RS flip-flop
   END_IF;
   IF #Rd.StatWord.Warning AND #Mot.comOk AND #area THEN #war := TRUE; END_IF;
END_REGION

REGION Network 36: fault motor protection motor
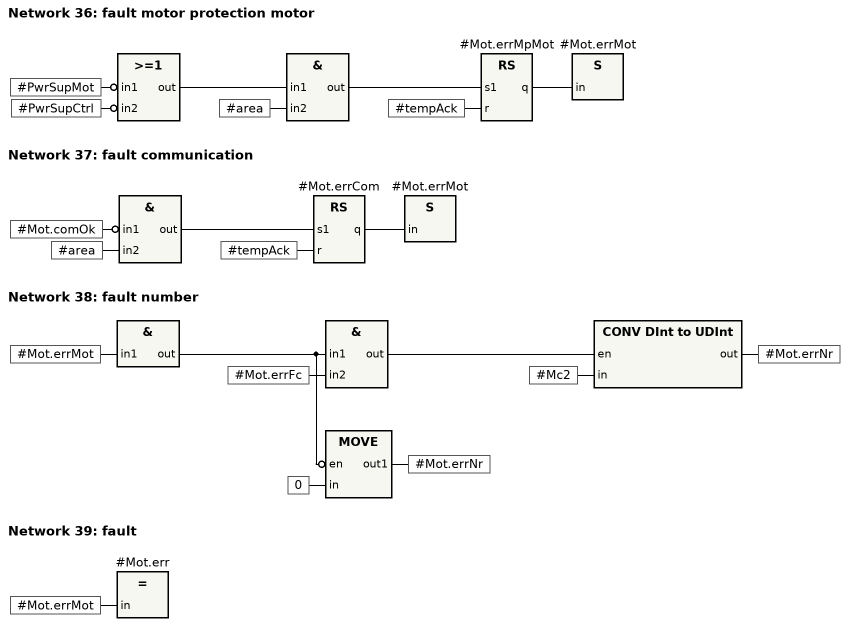
   IF #tempAck THEN
       #Mot.errMpMot := FALSE;   // RS flip-flop
   END_IF;
   IF (NOT #PwrSupMot OR NOT #PwrSupCtrl) AND #area THEN #Mot.errMpMot := TRUE; END_IF;
   IF #Mot.errMpMot THEN #Mot.errMot := TRUE; END_IF;
END_REGION

REGION Network 37: fault communication
   IF #tempAck THEN
       #Mot.errCom := FALSE;   // RS flip-flop
   END_IF;
   IF NOT #Mot.comOk AND #area THEN #Mot.errCom := TRUE; END_IF;
   IF #Mot.errCom THEN #Mot.errMot := TRUE; END_IF;
END_REGION

REGION Network 38: fault number
   IF #Mot.errMot AND #Mot.errFc THEN #Mot.errNr := DINT_TO_UDINT(#Mc2); END_IF;
   IF NOT #Mot.errMot THEN #Mot.errNr := 0; END_IF;
END_REGION

REGION Network 39: fault
   #Mot.err := #Mot.errMot;
END_REGION

REGION Network 40 (SCL): write outputs
   #comOk := #Mot.comOk;
   #ready := #Mot.ready;
   #err := #Mot.err;
   #errEnc := #Mot.err;
   #refOk := #Rd.StatWord.Homed;
   #refRun := #Sd.Ctrl.Home;
   #posOk := (#Rd.StatWord.InTargetPosition OR TRUE) AND #PosTolOk;
END_REGION

REGION Network 41 (SCL): in/out data
   #Mot.run := #Mot.plus OR #Mot.minus;
   #Mot.runDel := #Mot.plusDel OR #Mot.minusDel;
   #Mot.enStartP := false;
   #Mot.enStartM := false;
   #Mot.speedTar := DINT_TO_INT(#speed);
   #Mot.area := #area;

   IF #auto AND NOT #autoOld THEN
       #Mot.Hmi.man := false;
       #Mot.Hmi.manP := false;
       #Mot.Hmi.manM := false;
   END_IF;
   #autoOld := #auto;
END_REGION
END_FUNCTION_BLOCK

FUNCTION_BLOCK "SysPnSlaveDeactivate"   // FB2500, FBD
TITLE = Profinet Slave Deactivate / manage a sensor
{ S7_Optimized_Access := 'TRUE' }
AUTHOR : MiCROTEC
VERSION : 1.5
// -2018.12 : Martin
// stored: AutoNumber false, MemoryReserve 100, SetENOAutomatically false
   VAR_INPUT
      iSlave { ExternalAccessible := 'False'; ExternalVisible := 'False'; ExternalWritable := 'False'} : HW_DEVICE;
      iDeactivate { ExternalAccessible := 'False'; ExternalVisible := 'False'; ExternalWritable := 'False'} : Bool;
   END_VAR
   VAR_OUTPUT
      oSlaveActive { ExternalAccessible := 'False'; ExternalVisible := 'False'; ExternalWritable := 'False'} : Bool;   // Sensor fault , sensor is broken or is dirty
      oError { ExternalAccessible := 'False'; ExternalVisible := 'False'; ExternalWritable := 'False'} : Bool;   // Sensor fault , was to long occupied, maybe dirty or misaligned
   END_VAR
   VAR
      var { ExternalAccessible := 'False'; ExternalVisible := 'False'; ExternalWritable := 'False'} : Struct
         "bool" : Bool;
         "byte" : Byte;
         "word" : Word;
         "dword" : DWord;
         "int" : Int;
         "dint" : DInt;
         "real" : Real;
         s5time : S5Time;
         "time" : Time;
         hm : Array[1..16] of Bool;
         fm : Array[1..16] of Bool;
      END_STRUCT;
      vInit { ExternalAccessible := 'False'; ExternalVisible := 'False'; ExternalWritable := 'False'} : Bool;
      vStart { ExternalAccessible := 'False'; ExternalVisible := 'False'; ExternalWritable := 'False'} : Bool;
      vBusy { ExternalAccessible := 'False'; ExternalVisible := 'False'; ExternalWritable := 'False'} : Bool;
      vMode { ExternalAccessible := 'False'; ExternalVisible := 'False'; ExternalWritable := 'False'} : USInt;   // // 0: Status 1: aktivieren 2: deaktivieren
      vStep { ExternalAccessible := 'False'; ExternalVisible := 'False'; ExternalWritable := 'False'} : Int;
      vRetval { ExternalAccessible := 'False'; ExternalVisible := 'False'; ExternalWritable := 'False'} : Word;
   END_VAR
BEGIN

REGION Network 1 (SCL)
   CASE #vStep OF
       0:(*Init*)
           IF NOT #vInit OR #oError THEN
               #vStep := 110;
           ELSIF #oSlaveActive <> NOT #iDeactivate THEN
               #vStep := 10;
           END_IF;

       10:(*Aktiviere/Deaktiviere Slave*)
           #vStart := true;
           IF #iDeactivate THEN
               #vMode := 2;
           ELSE
               #vMode := 1;
           END_IF;
           #vStep := 20;

       20:(*Warte bis Fertig*)
           IF NOT #vBusy THEN
               #vStep := 30;
           END_IF;

       30:(*fertig*)
           #oError := #vRetval >= W#16#8000;
           #vStart := FALSE;
           #vStep := 110;

       110: (*Status holen*)
           #vStart := true;
           #vMode := 0;
           #vStep := 120;

       120:(*Warte bis Fertig*)
           IF NOT #vBusy THEN
               #vStep := 130;
           END_IF;

       130:(*fertig*)
           #oSlaveActive := #vRetval = 1;
           #oError := #vRetval >= W#16#8000;
           #vStart := FALSE;
           #vInit := true;
           #vStep := 0;


   END_CASE;

   #vRetval := D_ACT_DP(REQ := #vStart, MODE := #vMode, LADDR := #iSlave, BUSY => #vBusy);
END_REGION
END_FUNCTION_BLOCK

FUNCTION_BLOCK "AdjLeft"   // FB525, FBD
{ S7_Optimized_Access := 'TRUE' }
// stored: AutoNumber false, MemoryReserve 100, SetENOAutomatically false
   VAR
      Var { ExternalAccessible := 'False'; ExternalVisible := 'False'; ExternalWritable := 'False'} : "TypeVar";
      Cmd { ExternalAccessible := 'False'; ExternalVisible := 'False'; ExternalWritable := 'False'} : "TypeCmd";
      Enc { ExternalAccessible := 'False'; ExternalVisible := 'False'; ExternalWritable := 'False'} : "SysCounterFast";
      Pos { ExternalAccessible := 'False'; ExternalVisible := 'False'; ExternalWritable := 'False'} : "SysPos";
      AdjSlow { ExternalAccessible := 'False'; ExternalVisible := 'False'; ExternalWritable := 'False'} : "SysMotor";
      AdjFast { ExternalAccessible := 'False'; ExternalVisible := 'False'; ExternalWritable := 'False'} : "SysLinMotC1150";
      TAutoOn { ExternalAccessible := 'False'; ExternalVisible := 'False'; ExternalWritable := 'False'} : TON_TIME;
      TAutoTarPosManOn { ExternalAccessible := 'False'; ExternalVisible := 'False'; ExternalWritable := 'False'} : TON_TIME;
      T { ExternalAccessible := 'False'; ExternalVisible := 'False'; ExternalWritable := 'False'} : Array[1..5] of IEC_TIMER;
      adjFastPnSlaveOff { ExternalAccessible := 'False'; ExternalVisible := 'False'; ExternalWritable := 'False'} : "SysPnSlaveDeactivate";
      tarOld { ExternalAccessible := 'False'; ExternalVisible := 'False'; ExternalWritable := 'False'} : DInt;
      autoTarPosMan { ExternalAccessible := 'False'; ExternalVisible := 'False'; ExternalWritable := 'False'} : Bool;
      setValueEnc { ExternalAccessible := 'False'; ExternalVisible := 'False'; ExternalWritable := 'False'} : Bool;
      autoRef { ExternalAccessible := 'False'; ExternalVisible := 'False'; ExternalWritable := 'False'} : Bool;
      posOld { ExternalAccessible := 'False'; ExternalVisible := 'False'; ExternalWritable := 'False'} : Real;
      posDiff { ExternalAccessible := 'False'; ExternalVisible := 'False'; ExternalWritable := 'False'} : Real;
   END_VAR
   VAR_TEMP
      CtrlPc : Struct
         ackErr : Bool;
         manModeActive : Bool;
         manP : Bool;
         manM : Bool;
         manRefRun : Bool;
      END_STRUCT;
      CtrlLinMot : Struct
         mode : Int;
         target : Real;
         acc : Real;
         dec : Real;
         jerk : Real;
         speed : Real;
      END_STRUCT;
      refPosDiff : DInt;
      offsetNoStd : Real;
      refPosDiffCalib : DInt;
      modeCalib : Int;
      disMechanicToZero : Int;   // distance mechanic part left to zero [mm]
   END_VAR
   VAR_TEMP   // added for the SCL form of the ladder/FBD networks
      _w1 : Bool;
   END_VAR
BEGIN

REGION Network 1 (SCL): offset for no standard calibration
   (* 
   normally the distance from camera TO board should be 550mm
   for special application the distance is different
   the distance can be changed in the goldeneye program
   if its different then 550mm a offset will be added
   *)
   #offsetNoStd := 0.0;
   IF "ComRd".Data.Left.RefPosToBoard <> 550 THEN
       #offsetNoStd := (DINT_TO_REAL("ComRd".Data.Left.RefPosToBoard) - 550.0);
   ELSE
       #offsetNoStd := 0.0;
   END_IF;
END_REGION

REGION Network 2 (SCL): calibration value for offset
   (* 
   modus for calibartion
   camera must be referenced first
   mode 1 -->   the camera must be moved manually to position 550mm from board and
                 then press "Set Nullpoint"
   mode 2 -->   the camera must be moved to a other position and
                 then must be measured from the calibration tool to the camera and
                 this value must be putted in after pressing "Set Nullpoint"
   *)     
   #disMechanicToZero := 870;  
   #modeCalib := 2;
   IF #modeCalib = 1 THEN
       #refPosDiffCalib := "ComRd".Data.Left.TargetPos;
   ELSIF #modeCalib = 2 THEN
       #refPosDiffCalib := (#disMechanicToZero * 10) - ("ComRd".Data.Left.CalibratePos + 5500);
   END_IF;
END_REGION

REGION Network 3 (SCL): calibration value from pc
   "ComSd".Data.Left.SetCalibratePosOk := FALSE;

   IF "ComRd".Data.Left.SetCalibratePos THEN

       IF "G".Cfg.adjLeftActive THEN
           #refPosDiff := REAL_TO_DINT("Enc"."8BC1.L".act * 10.0) - #refPosDiffCalib;
       ELSIF "G".Cfg.adjLeftActiveLinMot THEN
           #refPosDiff := REAL_TO_DINT("Enc"."8U1.L".act * 10.0) - #refPosDiffCalib;
       END_IF;

       "Ref".adjLeftCalOffset := #refPosDiff;
       "ComSd".Data.Left.SetCalibratePosOk := TRUE;

   END_IF;
END_REGION

REGION Network 4 (SCL): target position
   #Cmd.target := "G".Batch.width / 2.0;
   IF "G".Cfg.modeBoardPassing = 2 AND ("G".Cfg.modeDimension = 2 OR "G".Cfg.modeDimension = 4) AND NOT "G".Batch.stdActive THEN
       #Cmd.target := "G".Batch.width / 2.0 + ("G".Batch.widthMeasure - "G".Batch.width);
   END_IF;

   IF "G".Cfg.modeBoardPassing = 3 AND ("G".Cfg.modeDimension = 2 OR "G".Cfg.modeDimension = 4) AND NOT "G".Batch.stdActive THEN
       #Cmd.target := "G".Batch.senLeftVal;
   END_IF;

   IF #autoTarPosMan THEN
       #Cmd.target := DINT_TO_REAL(("ComRd".Data.Left.TargetPos)) / 10.0;
   END_IF;

   "Ref".adjLeftTar := #Cmd.target + (DINT_TO_REAL("Ref".adjLeftCalOffset) / 10.0) + #offsetNoStd + "Enc"."8B1.B".offset;
END_REGION

REGION Network 5 (SCL): data from pc
   IF NOT "G".errComPc THEN
       #CtrlPc.manModeActive := "ComRd".Data.Left.ManModeActive;
       #CtrlPc.manP := "ComRd".Data.Left.ManPlus;
       #CtrlPc.manM := "ComRd".Data.Left.ManMinus;
       #CtrlPc.manRefRun := "ComRd".Data.Left.ManRefRun;
   ELSE
       #CtrlPc.manModeActive := TRUE;
       #CtrlPc.manP := FALSE;
       #CtrlPc.manM := FALSE;
       #CtrlPc.manRefRun := FALSE;
   END_IF;
   #CtrlPc.ackErr := "G".ack;
END_REGION

REGION Network 6: off
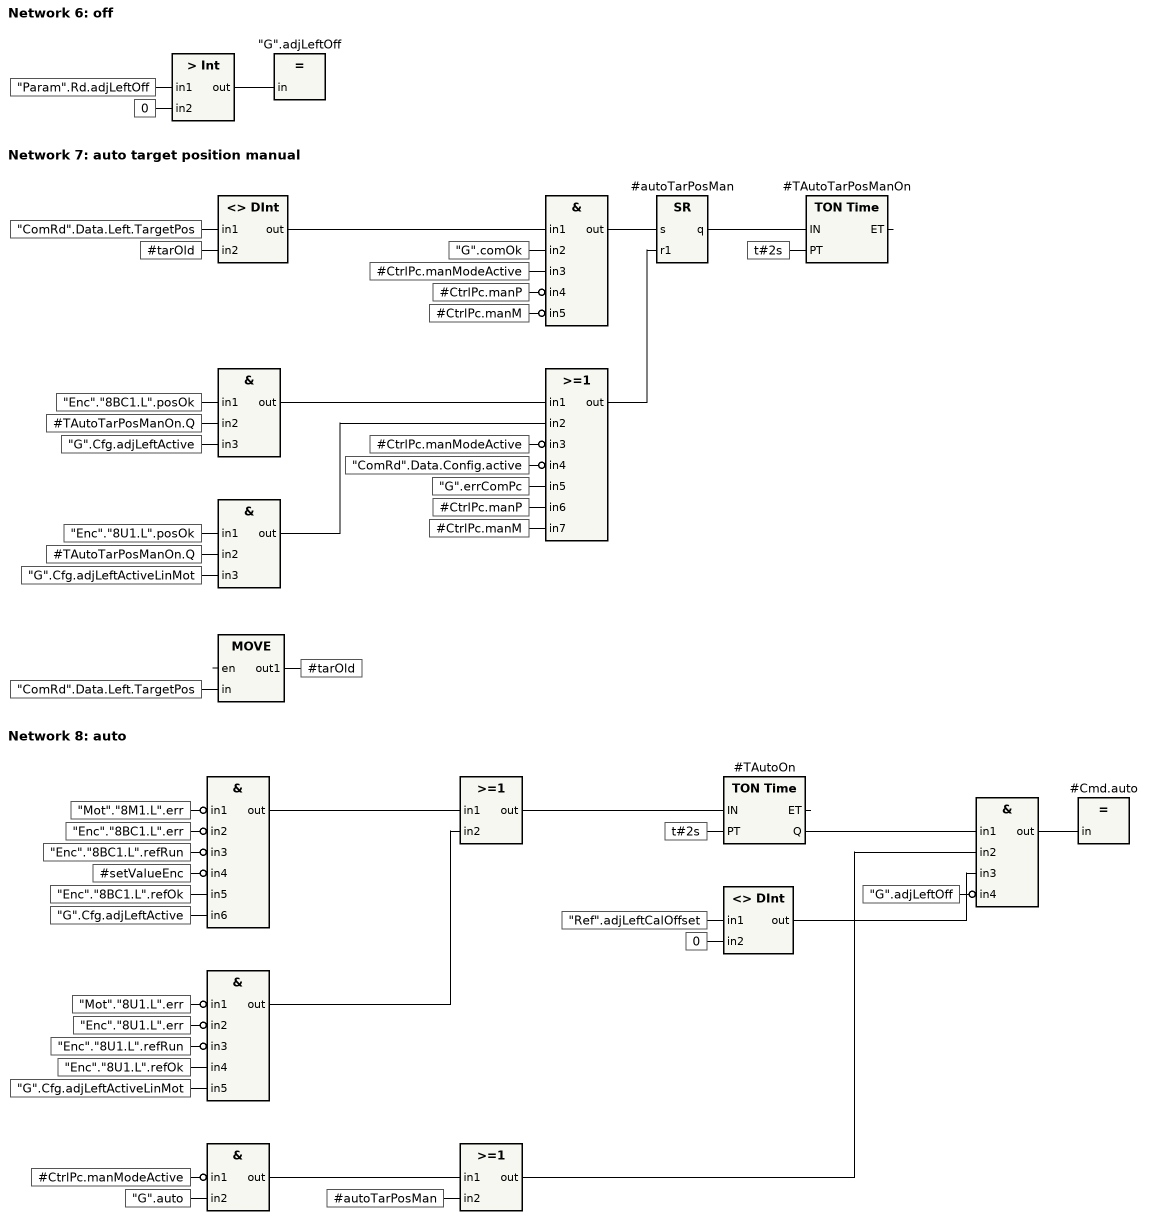
   "G".adjLeftOff := "Param".Rd.adjLeftOff > 0;
END_REGION

REGION Network 7: auto target position manual
   IF ("ComRd".Data.Left.TargetPos <> #tarOld) AND "G".comOk AND #CtrlPc.manModeActive AND NOT #CtrlPc.manP AND NOT #CtrlPc.manM THEN
       #autoTarPosMan := TRUE;   // SR flip-flop
   END_IF;
   IF ("Enc"."8BC1.L".posOk AND #TAutoTarPosManOn.Q AND "G".Cfg.adjLeftActive) OR ("Enc"."8U1.L".posOk AND #TAutoTarPosManOn.Q AND "G".Cfg.adjLeftActiveLinMot) OR NOT #CtrlPc.manModeActive OR NOT "ComRd".Data.Config.active OR "G".errComPc OR #CtrlPc.manP OR #CtrlPc.manM THEN
       #autoTarPosMan := FALSE;
   END_IF;
   #TAutoTarPosManOn(IN := #autoTarPosMan, PT := t#2s);   // TON
   #tarOld := "ComRd".Data.Left.TargetPos;
END_REGION

REGION Network 8: auto
   #TAutoOn(IN := (NOT "Mot"."8M1.L".err AND NOT "Enc"."8BC1.L".err AND NOT "Enc"."8BC1.L".refRun AND NOT #setValueEnc AND "Enc"."8BC1.L".refOk AND "G".Cfg.adjLeftActive) OR (NOT "Mot"."8U1.L".err AND NOT "Enc"."8U1.L".err AND NOT "Enc"."8U1.L".refRun AND "Enc"."8U1.L".refOk AND "G".Cfg.adjLeftActiveLinMot),   // TON
            PT := t#2s);
   #Cmd.auto := #TAutoOn.Q AND ((NOT #CtrlPc.manModeActive AND "G".auto) OR #autoTarPosMan) AND ("Ref".adjLeftCalOffset <> 0) AND NOT "G".adjLeftOff;
END_REGION

REGION Network 9: manual
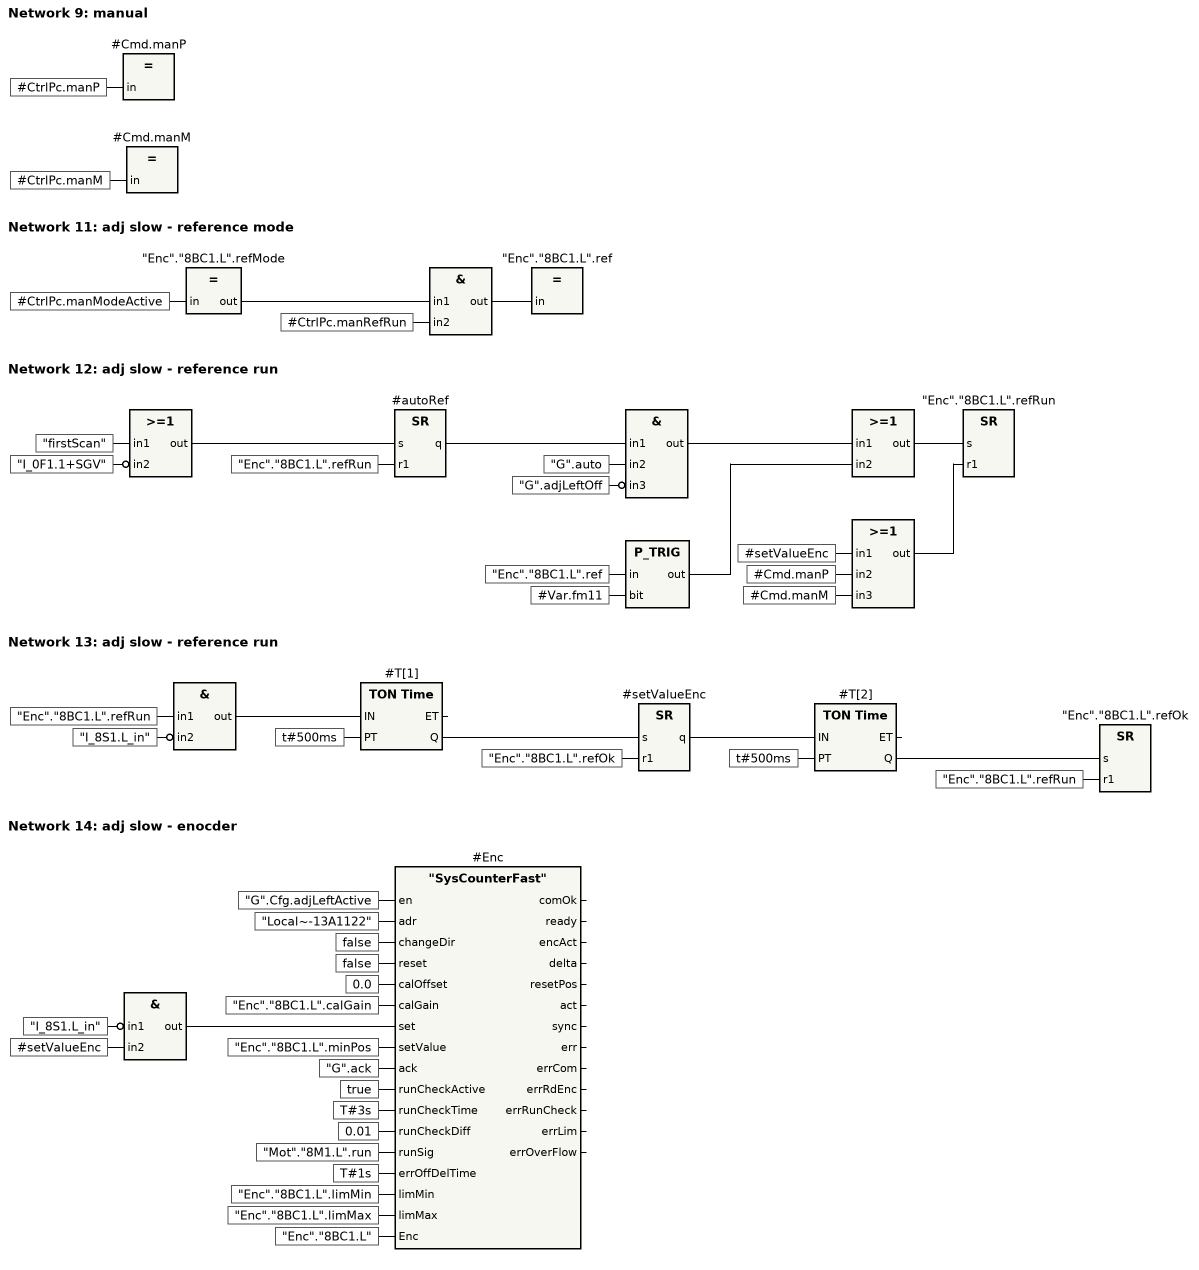
   #Cmd.manP := #CtrlPc.manP;
   #Cmd.manM := #CtrlPc.manM;
END_REGION

REGION Network 10 (SCL): adj slow - calibration value
   "Enc"."8BC1.L".calGain := -0.0275;

   "Enc"."8BC1.L".minPos := 10.0;
   "Enc"."8BC1.L".maxPos := 210.0;

   "Enc"."8BC1.L".limMin := "Enc"."8BC1.L".minPos - 5.0;
   "Enc"."8BC1.L".limMax := "Enc"."8BC1.L".maxPos + 5.0;

   "Enc"."8BC1.L".tarMinPos := "Enc"."8BC1.L".minPos + 0.0;
   "Enc"."8BC1.L".tarMaxPos := "Enc"."8BC1.L".maxPos - 0.0;
END_REGION

REGION Network 11: adj slow - reference mode
   "Enc"."8BC1.L".refMode := #CtrlPc.manModeActive;
   "Enc"."8BC1.L".ref := #CtrlPc.manModeActive AND #CtrlPc.manRefRun;
END_REGION

REGION Network 12: adj slow - reference run
   IF "firstScan" OR NOT "I_0F1.1+SGV" THEN
       #autoRef := TRUE;   // SR flip-flop
   END_IF;
   IF "Enc"."8BC1.L".refRun THEN #autoRef := FALSE; END_IF;
   #_w1 := "Enc"."8BC1.L".ref AND NOT #Var.fm11;   // rising edge
   #Var.fm11 := "Enc"."8BC1.L".ref;
   IF (#autoRef AND "G".auto AND NOT "G".adjLeftOff) OR #_w1 THEN
       "Enc"."8BC1.L".refRun := TRUE;   // SR flip-flop
   END_IF;
   IF #setValueEnc OR #Cmd.manP OR #Cmd.manM THEN "Enc"."8BC1.L".refRun := FALSE; END_IF;
END_REGION

REGION Network 13: adj slow - reference run
   #T[1].TON(IN := "Enc"."8BC1.L".refRun AND NOT "I_8S1.L_in", PT := t#500ms);
   IF #T[1].Q THEN
       #setValueEnc := TRUE;   // SR flip-flop
   END_IF;
   IF "Enc"."8BC1.L".refOk THEN #setValueEnc := FALSE; END_IF;
   #T[2].TON(IN := #setValueEnc, PT := t#500ms);
   IF #T[2].Q THEN
       "Enc"."8BC1.L".refOk := TRUE;   // SR flip-flop
   END_IF;
   IF "Enc"."8BC1.L".refRun THEN "Enc"."8BC1.L".refOk := FALSE; END_IF;
END_REGION

REGION Network 14: adj slow - enocder
   IF "G".Cfg.adjLeftActive THEN
       #Enc(adr := "Local~-13A1122",   // "SysCounterFast"
            changeDir := false,
            reset := false,
            calOffset := 0.0,
            calGain := "Enc"."8BC1.L".calGain,
            set := NOT "I_8S1.L_in" AND #setValueEnc,
            setValue := "Enc"."8BC1.L".minPos,
            ack := "G".ack,
            runCheckActive := true,
            runCheckTime := T#3s,
            runCheckDiff := 0.01,
            runSig := "Mot"."8M1.L".run,
            errOffDelTime := T#1s,
            limMin := "Enc"."8BC1.L".limMin,
            limMax := "Enc"."8BC1.L".limMax,
            Enc := "Enc"."8BC1.L");
   END_IF;
END_REGION

REGION Network 15: adj slow - pos
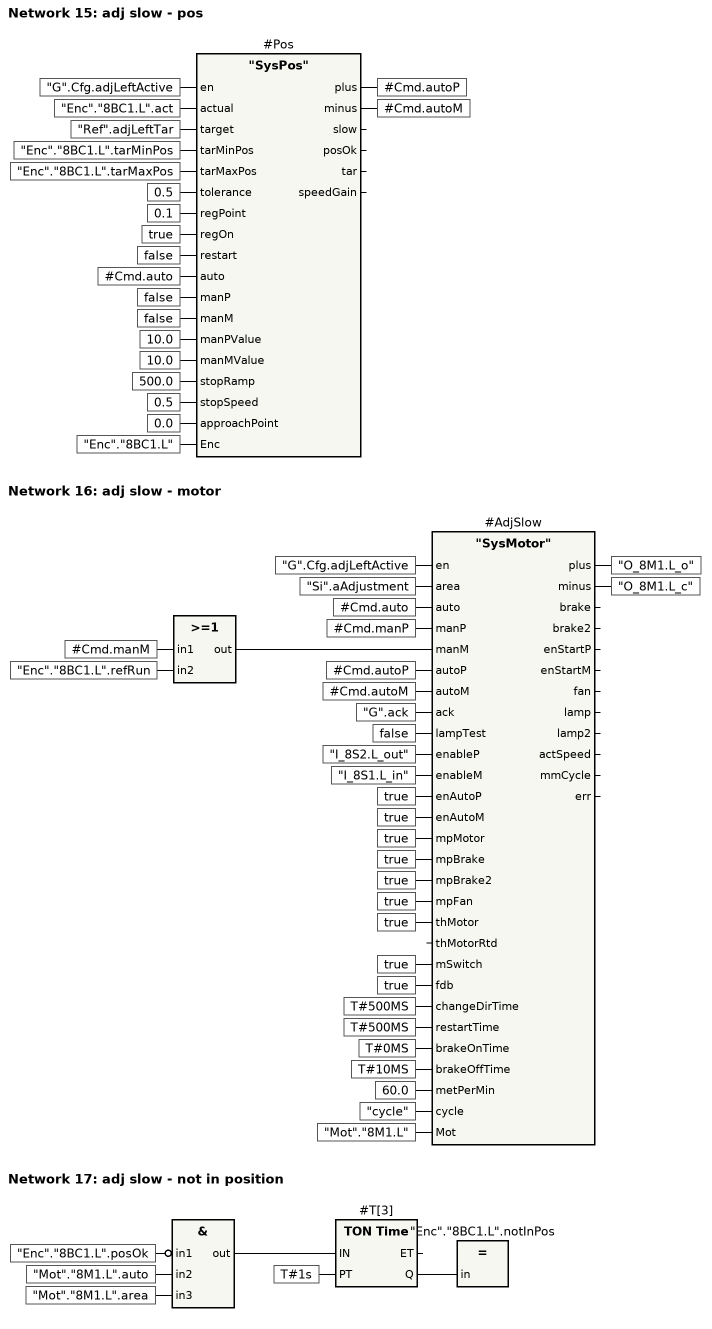
   IF "G".Cfg.adjLeftActive THEN
       #Pos(actual := "Enc"."8BC1.L".act,   // "SysPos"
            target := "Ref".adjLeftTar,
            tarMinPos := "Enc"."8BC1.L".tarMinPos,
            tarMaxPos := "Enc"."8BC1.L".tarMaxPos,
            tolerance := 0.5,
            regPoint := 0.1,
            regOn := true,
            restart := false,
            auto := #Cmd.auto,
            manP := false,
            manM := false,
            manPValue := 10.0,
            manMValue := 10.0,
            stopRamp := 500.0,
            stopSpeed := 0.5,
            approachPoint := 0.0,
            Enc := "Enc"."8BC1.L",
            plus => #Cmd.autoP,
            minus => #Cmd.autoM);
   END_IF;
END_REGION

REGION Network 16: adj slow - motor
   IF "G".Cfg.adjLeftActive THEN
       #AdjSlow(area := "Si".aAdjustment,   // "SysMotor"
                auto := #Cmd.auto,
                manP := #Cmd.manP,
                manM := #Cmd.manM OR "Enc"."8BC1.L".refRun,
                autoP := #Cmd.autoP,
                autoM := #Cmd.autoM,
                ack := "G".ack,
                lampTest := false,
                enableP := "I_8S2.L_out",
                enableM := "I_8S1.L_in",
                enAutoP := true,
                enAutoM := true,
                mpMotor := true,
                mpBrake := true,
                mpBrake2 := true,
                mpFan := true,
                thMotor := true,
                mSwitch := true,
                fdb := true,
                changeDirTime := T#500MS,
                restartTime := T#500MS,
                brakeOnTime := T#0MS,
                brakeOffTime := T#10MS,
                metPerMin := 60.0,
                cycle := "cycle",
                Mot := "Mot"."8M1.L",
                plus => "O_8M1.L_o",
                minus => "O_8M1.L_c");
   END_IF;
END_REGION

REGION Network 17: adj slow - not in position
   #T[3].TON(IN := NOT "Enc"."8BC1.L".posOk AND "Mot"."8M1.L".auto AND "Mot"."8M1.L".area, PT := T#1s);
   "Enc"."8BC1.L".notInPos := #T[3].Q;
END_REGION

REGION Network 18: adj slow - sensor monitoring
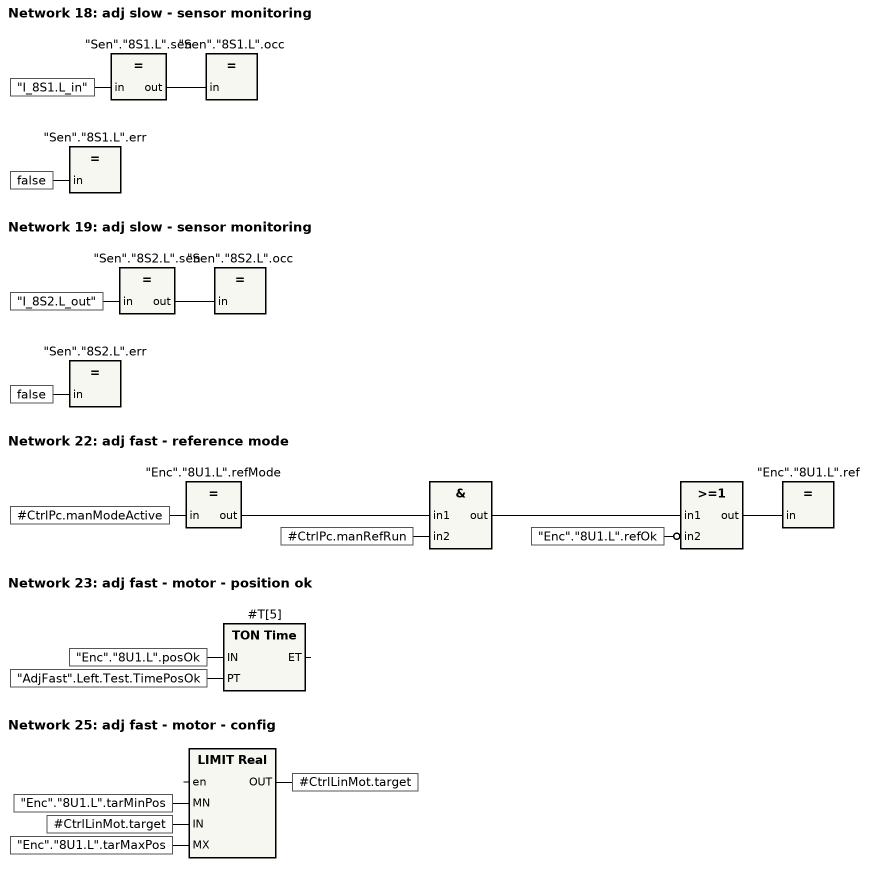
   "Sen"."8S1.L".sen := "I_8S1.L_in";
   "Sen"."8S1.L".occ := "I_8S1.L_in";
   "Sen"."8S1.L".err := false;
END_REGION

REGION Network 19: adj slow - sensor monitoring
   "Sen"."8S2.L".sen := "I_8S2.L_out";
   "Sen"."8S2.L".occ := "I_8S2.L_out";
   "Sen"."8S2.L".err := false;
END_REGION

REGION Network 21 (SCL): adj fast - calibration value
   "Enc"."8U1.L".calGain := 1.0;

   "Enc"."8U1.L".minPos := 5.0;
   "Enc"."8U1.L".maxPos := 155.0;

   "Enc"."8U1.L".limMin := "Enc"."8U1.L".minPos - 5.0;
   "Enc"."8U1.L".limMax := "Enc"."8U1.L".maxPos + 5.0;

   "Enc"."8U1.L".tarMinPos := "Enc"."8U1.L".minPos + 0.0;
   "Enc"."8U1.L".tarMaxPos := "Enc"."8U1.L".maxPos - 0.0;
END_REGION

REGION Network 22: adj fast - reference mode
   "Enc"."8U1.L".refMode := #CtrlPc.manModeActive;
   "Enc"."8U1.L".ref := (#CtrlPc.manModeActive AND #CtrlPc.manRefRun) OR NOT "Enc"."8U1.L".refOk;
END_REGION

REGION Network 23: adj fast - motor - position ok
   #T[5].TON(IN := "Enc"."8U1.L".posOk, PT := "AdjFast".Left.Test.TimePosOk);
END_REGION

REGION Network 24 (SCL): adj fast - motor - config

   //############################################################
   // min            5     mm
   // max          155     mm

   // speed        02      m/s
   // acc/dec      24      m/s2
   // jerk         450     m/s3

   // mode         BestehornVAJ
   //############################################################

   // only testmode for plc
   IF "AdjFast".Left.Test.ModeActive AND NOT #CtrlPc.manModeActive THEN
       IF "AdjFast".Left.Test.TarPos = "AdjFast".Left.Test.TarPos1 AND #T[5].Q THEN
           "AdjFast".Left.Test.TarPos := "AdjFast".Left.Test.TarPos2;
       ELSIF "AdjFast".Left.Test.TarPos = "AdjFast".Left.Test.TarPos2 AND #T[5].Q THEN
           "AdjFast".Left.Test.TarPos := "AdjFast".Left.Test.TarPos1;
       END_IF;
       "Ref".adjLeftTar := "AdjFast".Left.Test.TarPos;
   END_IF;

   // active mode
   #CtrlLinMot.mode := 3;
   #CtrlLinMot.target := "Ref".adjLeftTar;
   #CtrlLinMot.speed := 2.0;
   #CtrlLinMot.acc := 24.0;
   #CtrlLinMot.dec := 0.0;
   #CtrlLinMot.jerk := 450.0;

   // only testmode for plc
   IF "AdjFast".Left.Mode = 1 THEN
       #CtrlLinMot.mode := 1;
       #CtrlLinMot.target := "AdjFast".Left.VAI.Par1;
       #CtrlLinMot.speed := "AdjFast".Left.VAI.Par2;
       #CtrlLinMot.acc := "AdjFast".Left.VAI.Par3;
       #CtrlLinMot.dec := "AdjFast".Left.VAI.Par4;
       #CtrlLinMot.jerk := 0.0;
   ELSIF "AdjFast".Left.Mode = 2 THEN
       #CtrlLinMot.mode := 2;
       #CtrlLinMot.target := "AdjFast".Left.SinVA.Par1;
       #CtrlLinMot.speed := "AdjFast".Left.SinVA.Par2;
       #CtrlLinMot.acc := "AdjFast".Left.SinVA.Par3;
       #CtrlLinMot.dec := 0.0;
       #CtrlLinMot.jerk := 0.0;
   ELSIF "AdjFast".Left.Mode = 3 THEN
       #CtrlLinMot.mode := 3;
       #CtrlLinMot.target := "AdjFast".Left.BestehornVAJ.Par1;
       #CtrlLinMot.speed := "AdjFast".Left.BestehornVAJ.Par2;
       #CtrlLinMot.acc := "AdjFast".Left.BestehornVAJ.Par3;
       #CtrlLinMot.dec := 0.0;
       #CtrlLinMot.jerk := "AdjFast".Left.BestehornVAJ.Par4;
   END_IF;
END_REGION

REGION Network 25: adj fast - motor - config
   #CtrlLinMot.target := LIMIT(MN := "Enc"."8U1.L".tarMinPos, IN := #CtrlLinMot.target, MX := "Enc"."8U1.L".tarMaxPos);
END_REGION

REGION Network 26: adj fast - motor
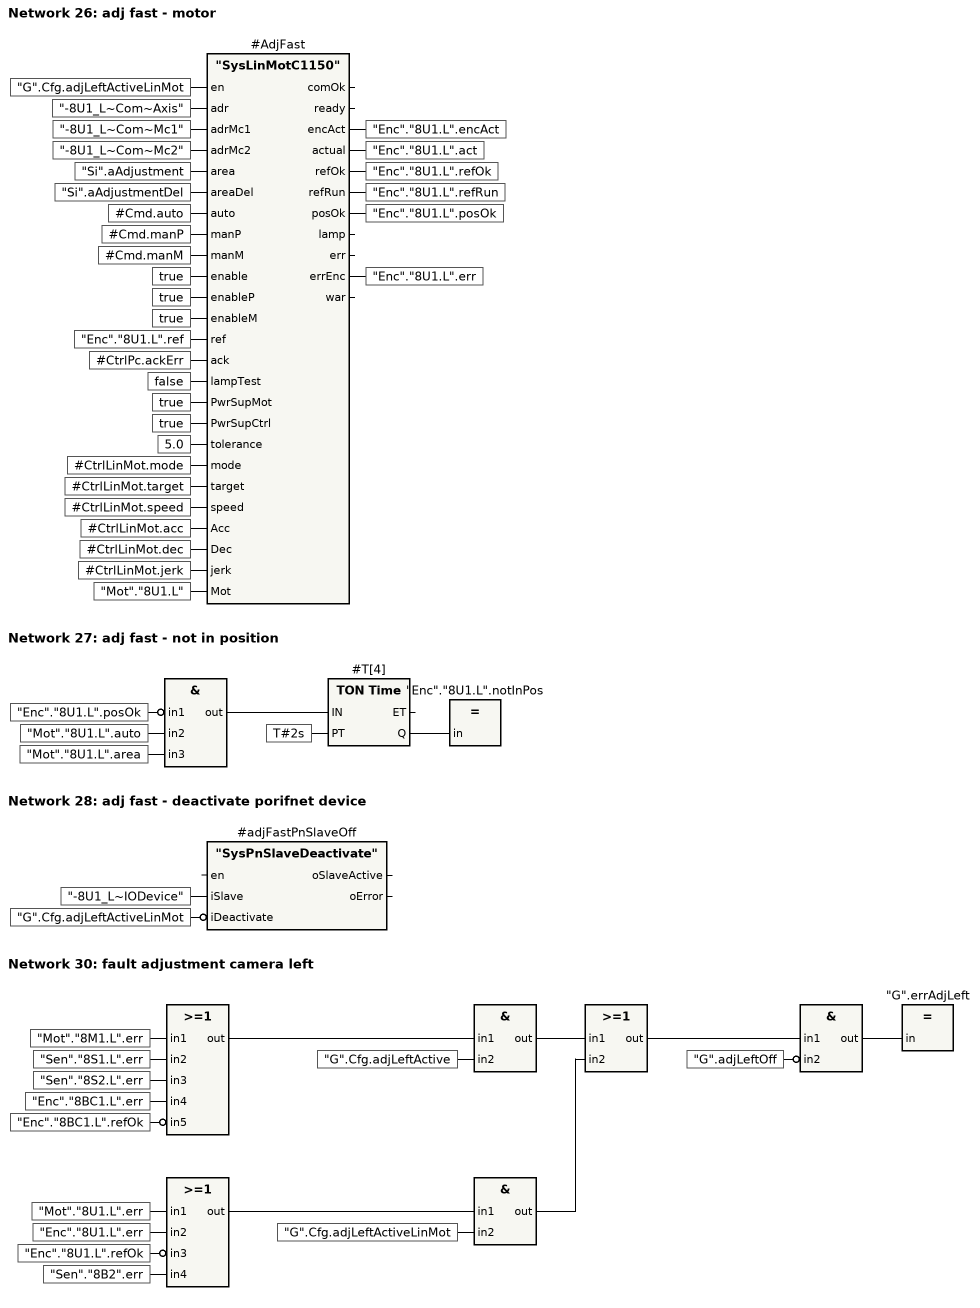
   IF "G".Cfg.adjLeftActiveLinMot THEN
       #AdjFast(adr := "-8U1_L~Com~Axis",   // "SysLinMotC1150"
                adrMc1 := "-8U1_L~Com~Mc1",
                adrMc2 := "-8U1_L~Com~Mc2",
                area := "Si".aAdjustment,
                areaDel := "Si".aAdjustmentDel,
                auto := #Cmd.auto,
                manP := #Cmd.manP,
                manM := #Cmd.manM,
                enable := true,
                enableP := true,
                enableM := true,
                ref := "Enc"."8U1.L".ref,
                ack := #CtrlPc.ackErr,
                lampTest := false,
                PwrSupMot := true,
                PwrSupCtrl := true,
                tolerance := 5.0,
                mode := #CtrlLinMot.mode,
                target := #CtrlLinMot.target,
                speed := #CtrlLinMot.speed,
                Acc := #CtrlLinMot.acc,
                Dec := #CtrlLinMot.dec,
                jerk := #CtrlLinMot.jerk,
                Mot := "Mot"."8U1.L",
                encAct => "Enc"."8U1.L".encAct,
                actual => "Enc"."8U1.L".act,
                refOk => "Enc"."8U1.L".refOk,
                refRun => "Enc"."8U1.L".refRun,
                posOk => "Enc"."8U1.L".posOk,
                errEnc => "Enc"."8U1.L".err);
   END_IF;
END_REGION

REGION Network 27: adj fast - not in position
   #T[4].TON(IN := NOT "Enc"."8U1.L".posOk AND "Mot"."8U1.L".auto AND "Mot"."8U1.L".area, PT := T#2s);
   "Enc"."8U1.L".notInPos := #T[4].Q;
END_REGION

REGION Network 28: adj fast - deactivate porifnet device
   #adjFastPnSlaveOff(iSlave := "-8U1_L~IODevice", iDeactivate := NOT "G".Cfg.adjLeftActiveLinMot);   // "SysPnSlaveDeactivate"
END_REGION

REGION Network 30: fault adjustment camera left
   "G".errAdjLeft := ((("Mot"."8M1.L".err OR "Sen"."8S1.L".err OR "Sen"."8S2.L".err OR "Enc"."8BC1.L".err OR NOT "Enc"."8BC1.L".refOk) AND "G".Cfg.adjLeftActive) OR (("Mot"."8U1.L".err OR "Enc"."8U1.L".err OR NOT "Enc"."8U1.L".refOk OR "Sen"."8B2".err) AND "G".Cfg.adjLeftActiveLinMot)) AND NOT "G".adjLeftOff;
END_REGION

REGION Network 31 (SCL): data to pc
   IF "G".Cfg.adjLeftActive THEN
       "Ref".adjLeftAct := REAL_TO_DINT("Enc"."8BC1.L".act * 10.0) - "Ref".adjLeftCalOffset - REAL_TO_DINT(#offsetNoStd * 10.0);
       "ComSd".Data.Left.ActualEncPos := REAL_TO_DINT("Enc"."8BC1.L".act * 10.0);
       "ComSd".Data.Left.ActualPos :=  "Ref".adjLeftAct;
       "ComSd".Data.Left.LimitSwitchMin := "Sen"."8S1.L".sen;
       "ComSd".Data.Left.LimitSwitchMax := "Sen"."8S2.L".sen;
       "ComSd".Data.Left.Err := "Mot"."8M1.L".err;
       "ComSd".Data.Left.ErrEnc := "Enc"."8BC1.L".err;
       "ComSd".Data.Left.PosOk := "Enc"."8BC1.L".posOk;
       "ComSd".Data.Left.Plus := "Mot"."8M1.L".plus;
       "ComSd".Data.Left.Minus := "Mot"."8M1.L".minus;
       "ComSd".Data.Left.refRun := "Enc"."8BC1.L".refRun;
       "ComSd".Data.Left.refOk := "Enc"."8BC1.L".refOk;
   ELSIF  "G".Cfg.adjLeftActiveLinMot THEN
       "Ref".adjLeftAct := REAL_TO_DINT("Enc"."8U1.L".act * 10.0) - "Ref".adjLeftCalOffset - REAL_TO_DINT(#offsetNoStd * 10.0);
       "ComSd".Data.Left.ActualEncPos := REAL_TO_DINT("Enc"."8U1.L".act * 10.0);
       "ComSd".Data.Left.ActualPos :=  "Ref".adjLeftAct;
       "ComSd".Data.Left.LimitSwitchMin := TRUE;
       "ComSd".Data.Left.LimitSwitchMax := TRUE;
       "ComSd".Data.Left.Err := "Mot"."8U1.L".err;
       "ComSd".Data.Left.ErrEnc := "Enc"."8U1.L".err;
       "ComSd".Data.Left.PosOk := "Enc"."8U1.L".posOk;
       "ComSd".Data.Left.Plus := "Mot"."8U1.L".plus;
       "ComSd".Data.Left.Minus := "Mot"."8U1.L".minus;
       "ComSd".Data.Left.refRun := "Enc"."8U1.L".refRun;
       "ComSd".Data.Left.refOk := "Enc"."8U1.L".refOk;
   ELSE
       "ComSd".Data.Left.ActualEncPos := 0;
       "ComSd".Data.Left.ActualPos := 0;
       "ComSd".Data.Left.LimitSwitchMin := FALSE;
       "ComSd".Data.Left.LimitSwitchMax := FALSE;
       "ComSd".Data.Left.Err := FALSE;
       "ComSd".Data.Left.ErrEnc := FALSE;
       "ComSd".Data.Left.PosOk := True;
       "ComSd".Data.Left.Plus := FALSE;
       "ComSd".Data.Left.Minus := FALSE;
       "ComSd".Data.Left.refRun := FALSE;
       "ComSd".Data.Left.refOk := TRUE;
   END_IF;
END_REGION

REGION Network 32: current monitoring - auto
